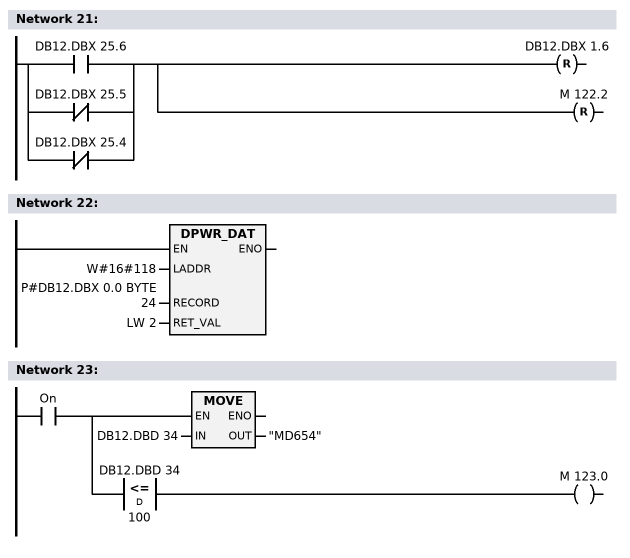
NETWORK
TITLE =
      O     DB12.DBX 25.6;
      ON    DB12.DBX 25.5;
      ON    DB12.DBX 25.4;
      R     DB12.DBX 1.6;
      R     M 122.2;
NETWORK
TITLE =
      CALL  "DPWR_DAT" (
           LADDR                    := W#16#118,
           RECORD                   := P#DB12.DBX 0.0 BYTE 24,
           RET_VAL                  := LW 2);
      NOP   0;
NETWORK
TITLE =
      A     "On";
      =     L 20.0;
      A     L 20.0;
      JNB   M019;
      L     DB12.DBD 34;
      T     "MD654";
M019: NOP   0;
      A     L 20.0;
      A(;
      L     DB12.DBD 34;
      L     100;
      <=D;
      );
      =     M 123.0;
END_FUNCTION

FUNCTION "FC50 - TEACH-IN" : VOID	// FC 50
VERSION : 0.1
BEGIN
// (block stored without names or comments; labels and parameter names are numbered)
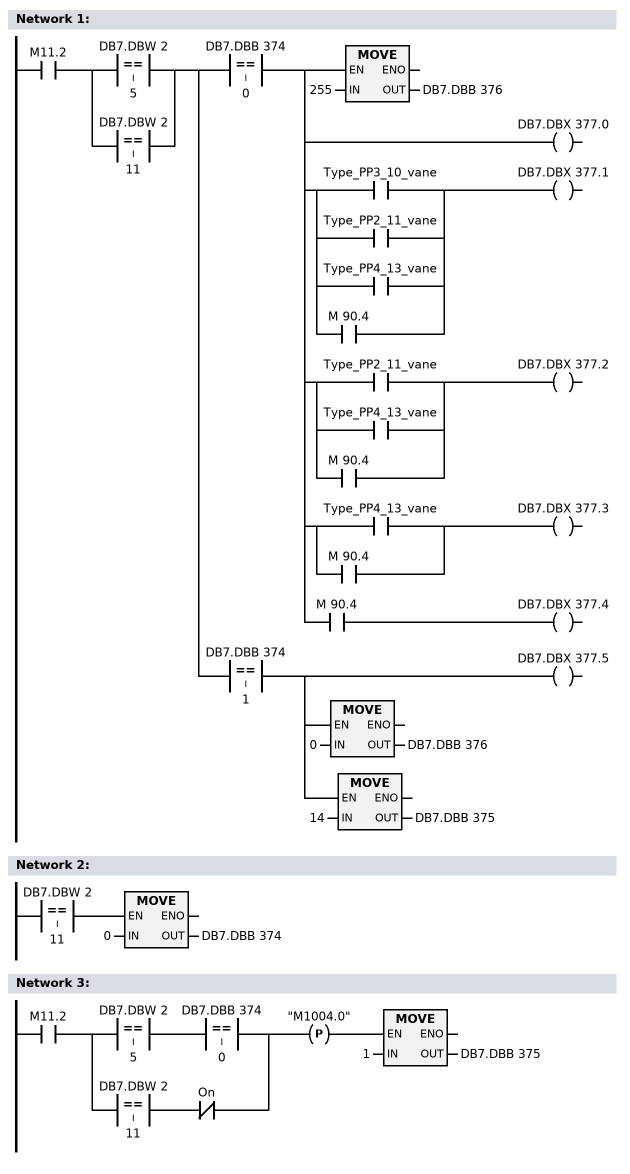
NETWORK
TITLE =
      A     "M11.2";
      A(;
      O(;
      L     DB7.DBW 2;
      L     5;
      ==I;
      );
      O(;
      L     DB7.DBW 2;
      L     11;
      ==I;
      );
      );
      =     L 8.0;
      A     L 8.0;
      A(;
      L     DB7.DBB 374;
      L     0;
      ==I;
      );
      =     L 8.1;
      A     L 8.1;
      JNB   M001;
      L     255;
      T     DB7.DBB 376;
M001: NOP   0;
      A     L 8.1;
      BLD   102;
      =     DB7.DBX 377.0;
      A     L 8.1;
      A(;
      O     "Type_PP3_10_vane";
      O     "Type_PP2_11_vane";
      O     "Type_PP4_13_vane";
      O     M 90.4;
      );
      =     DB7.DBX 377.1;
      A     L 8.1;
      A(;
      O     "Type_PP2_11_vane";
      O     "Type_PP4_13_vane";
      O     M 90.4;
      );
      =     DB7.DBX 377.2;
      A     L 8.1;
      A(;
      O     "Type_PP4_13_vane";
      O     M 90.4;
      );
      =     DB7.DBX 377.3;
      A     L 8.1;
      A     M 90.4;
      =     DB7.DBX 377.4;
      A     L 8.0;
      A(;
      L     DB7.DBB 374;
      L     1;
      ==I;
      );
      =     L 8.1;
      A     L 8.1;
      BLD   102;
      =     DB7.DBX 377.5;
      A     L 8.1;
      JNB   M002;
      L     0;
      T     DB7.DBB 376;
M002: NOP   0;
      A     L 8.1;
      JNB   M003;
      L     14;
      T     DB7.DBB 375;
M003: NOP   0;
NETWORK
TITLE =
      A(;
      L     DB7.DBW 2;
      L     11;
      ==I;
      );
      JNB   M004;
      L     0;
      T     DB7.DBB 374;
M004: NOP   0;
NETWORK
TITLE =
      A     "M11.2";
      A(;
      A(;
      L     DB7.DBW 2;
      L     5;
      ==I;
      );
      A(;
      L     DB7.DBB 374;
      L     0;
      ==I;
      );
      O;
      A(;
      L     DB7.DBW 2;
      L     11;
      ==I;
      );
      AN    "On";
      );
      FP    "M1004.0";
      JNB   M005;
      L     1;
      T     DB7.DBB 375;
M005: NOP   0;
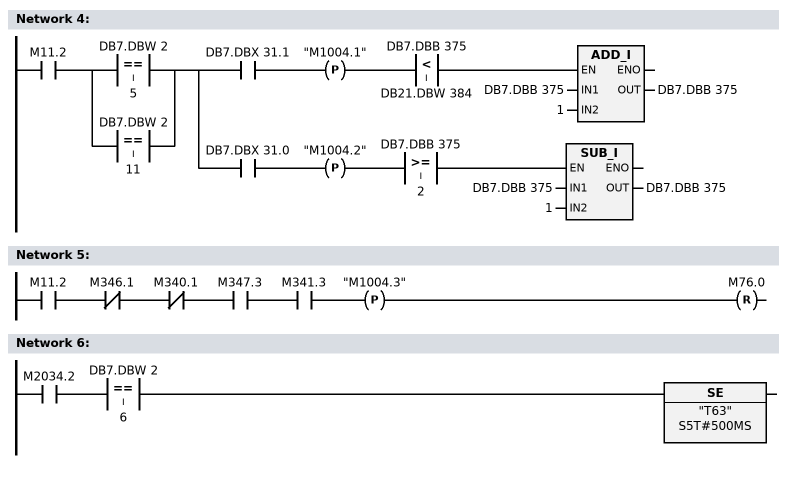
NETWORK
TITLE =
      A     "M11.2";
      A(;
      O(;
      L     DB7.DBW 2;
      L     5;
      ==I;
      );
      O(;
      L     DB7.DBW 2;
      L     11;
      ==I;
      );
      );
      =     L 8.0;
      A     L 8.0;
      A     DB7.DBX 31.1;
      FP    "M1004.1";
      A(;
      L     DB7.DBB 375;
      L     DB21.DBW 384;
      <I;
      );
      JNB   M006;
      L     DB7.DBB 375;
      L     1;
      +I;
      T     DB7.DBB 375;
M006: NOP   0;
      A     L 8.0;
      A     DB7.DBX 31.0;
      FP    "M1004.2";
      A(;
      L     DB7.DBB 375;
      L     2;
      >=I;
      );
      JNB   M007;
      L     DB7.DBB 375;
      L     1;
      -I;
      T     DB7.DBB 375;
M007: NOP   0;
NETWORK
TITLE =
      A     "M11.2";
      AN    "M346.1";
      AN    "M340.1";
      A     "M347.3";
      A     "M341.3";
      FP    "M1004.3";
      R     "M76.0";
NETWORK
TITLE =
      A     "M2034.2";
      A(;
      L     DB7.DBW 2;
      L     6;
      ==I;
      );
      L     S5T#500MS;
      SE    "T63";
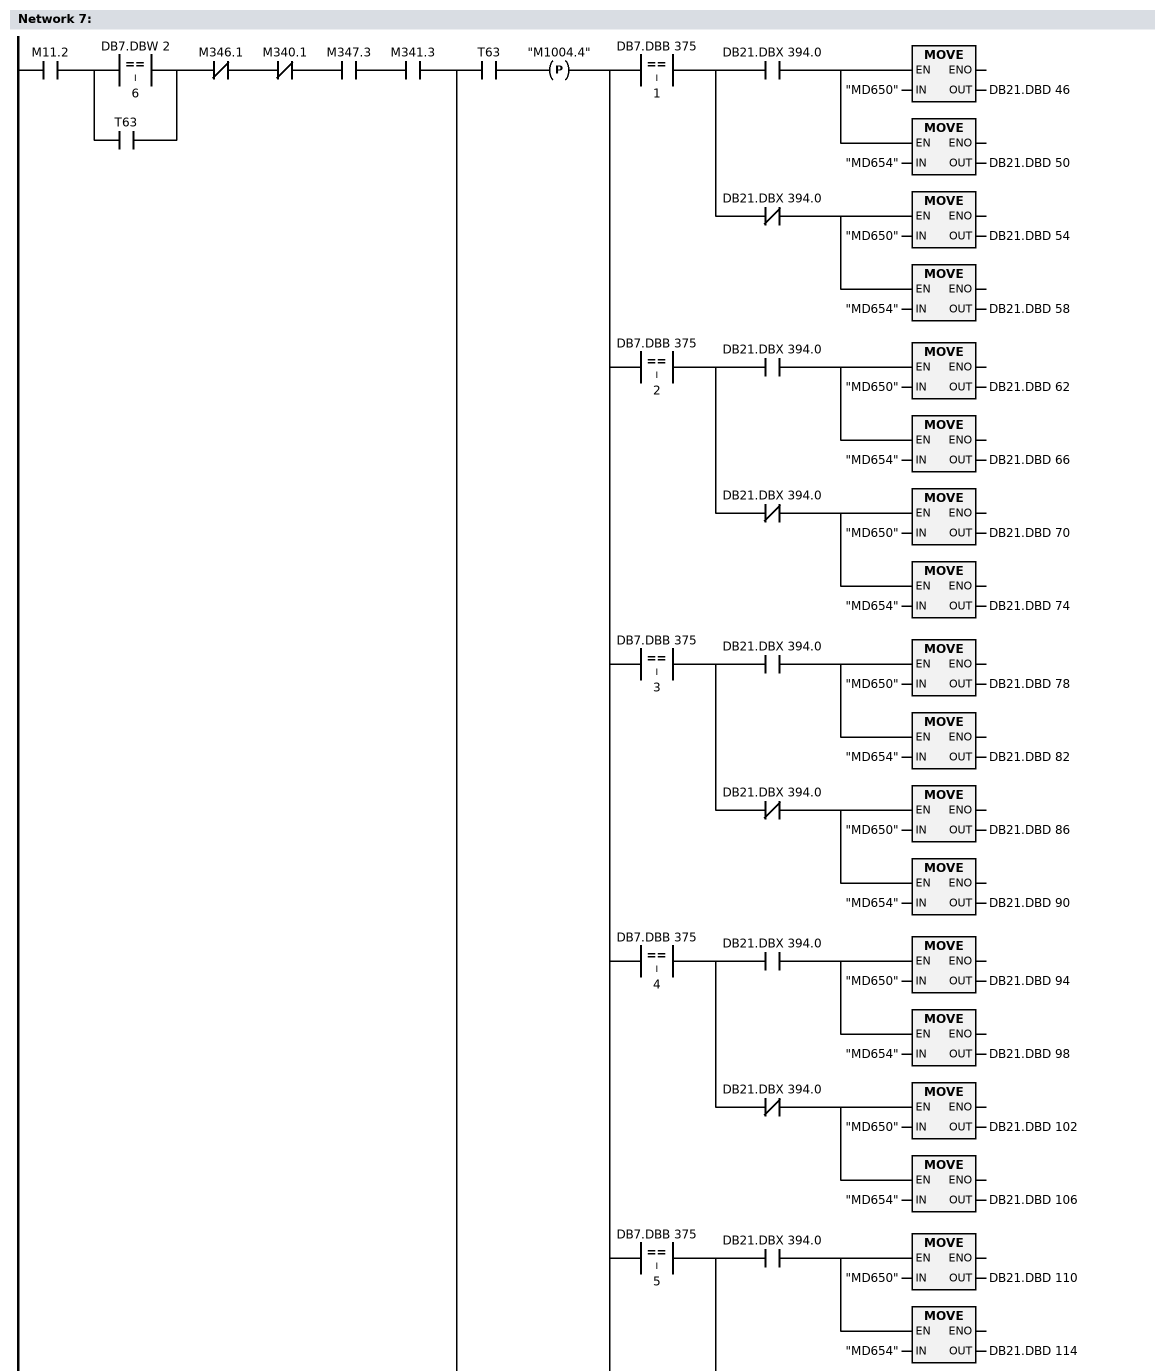
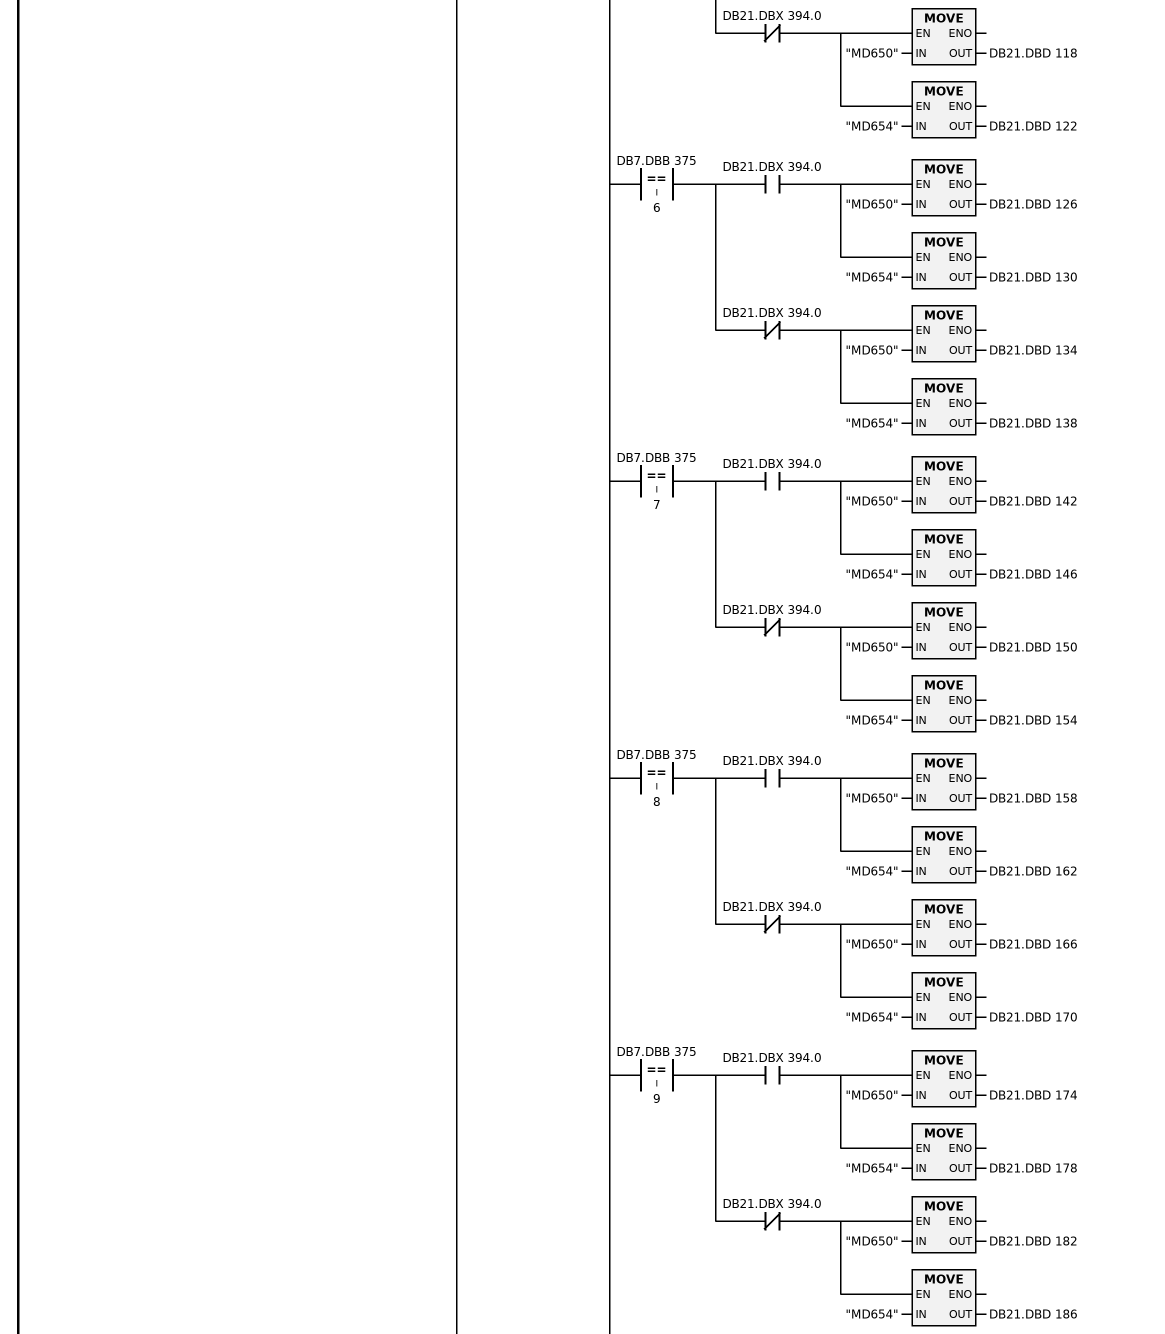
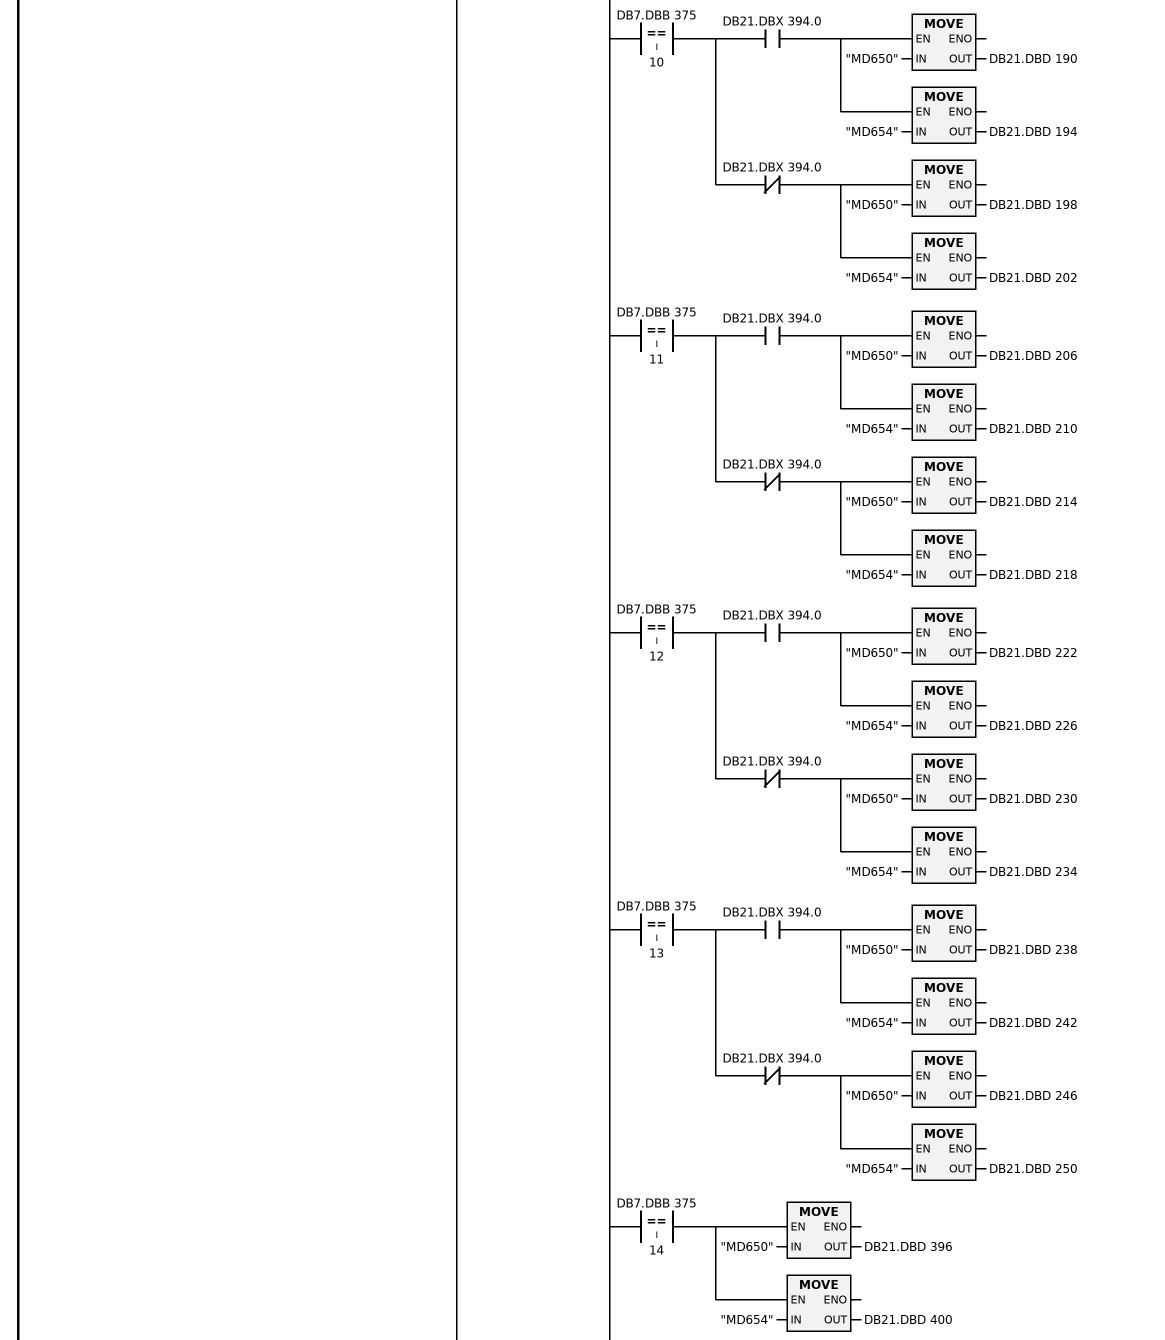
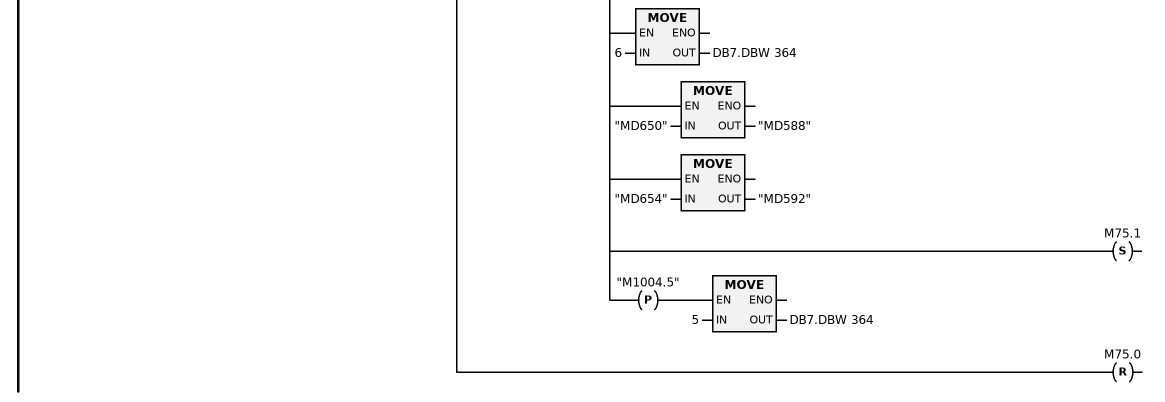
NETWORK
TITLE =
      A     "M11.2";
      A(;
      O(;
      L     DB7.DBW 2;
      L     6;
      ==I;
      );
      O     "T63";
      );
      AN    "M346.1";
      AN    "M340.1";
      A     "M347.3";
      A     "M341.3";
      =     L 8.0;
      A     L 8.0;
      A     "T63";
      FP    "M1004.4";
      =     L 8.1;
      A     L 8.1;
      A(;
      L     DB7.DBB 375;
      L     1;
      ==I;
      );
      =     L 8.2;
      A     L 8.2;
      A     DB21.DBX 394.0;
      =     L 8.3;
      A     L 8.3;
      JNB   M008;
      L     "MD650";
      T     DB21.DBD 46;
M008: NOP   0;
      A     L 8.3;
      JNB   M009;
      L     "MD654";
      T     DB21.DBD 50;
M009: NOP   0;
      A     L 8.2;
      AN    DB21.DBX 394.0;
      =     L 8.3;
      A     L 8.3;
      JNB   M010;
      L     "MD650";
      T     DB21.DBD 54;
M010: NOP   0;
      A     L 8.3;
      JNB   M011;
      L     "MD654";
      T     DB21.DBD 58;
M011: NOP   0;
      A     L 8.1;
      A(;
      L     DB7.DBB 375;
      L     2;
      ==I;
      );
      =     L 8.2;
      A     L 8.2;
      A     DB21.DBX 394.0;
      =     L 8.3;
      A     L 8.3;
      JNB   M012;
      L     "MD650";
      T     DB21.DBD 62;
M012: NOP   0;
      A     L 8.3;
      JNB   M013;
      L     "MD654";
      T     DB21.DBD 66;
M013: NOP   0;
      A     L 8.2;
      AN    DB21.DBX 394.0;
      =     L 8.3;
      A     L 8.3;
      JNB   M014;
      L     "MD650";
      T     DB21.DBD 70;
M014: NOP   0;
      A     L 8.3;
      JNB   M015;
      L     "MD654";
      T     DB21.DBD 74;
M015: NOP   0;
      A     L 8.1;
      A(;
      L     DB7.DBB 375;
      L     3;
      ==I;
      );
      =     L 8.2;
      A     L 8.2;
      A     DB21.DBX 394.0;
      =     L 8.3;
      A     L 8.3;
      JNB   M016;
      L     "MD650";
      T     DB21.DBD 78;
M016: NOP   0;
      A     L 8.3;
      JNB   M017;
      L     "MD654";
      T     DB21.DBD 82;
M017: NOP   0;
      A     L 8.2;
      AN    DB21.DBX 394.0;
      =     L 8.3;
      A     L 8.3;
      JNB   M018;
      L     "MD650";
      T     DB21.DBD 86;
M018: NOP   0;
      A     L 8.3;
      JNB   M019;
      L     "MD654";
      T     DB21.DBD 90;
M019: NOP   0;
      A     L 8.1;
      A(;
      L     DB7.DBB 375;
      L     4;
      ==I;
      );
      =     L 8.2;
      A     L 8.2;
      A     DB21.DBX 394.0;
      =     L 8.3;
      A     L 8.3;
      JNB   M020;
      L     "MD650";
      T     DB21.DBD 94;
M020: NOP   0;
      A     L 8.3;
      JNB   M021;
      L     "MD654";
      T     DB21.DBD 98;
M021: NOP   0;
      A     L 8.2;
      AN    DB21.DBX 394.0;
      =     L 8.3;
      A     L 8.3;
      JNB   M022;
      L     "MD650";
      T     DB21.DBD 102;
M022: NOP   0;
      A     L 8.3;
      JNB   M023;
      L     "MD654";
      T     DB21.DBD 106;
M023: NOP   0;
      A     L 8.1;
      A(;
      L     DB7.DBB 375;
      L     5;
      ==I;
      );
      =     L 8.2;
      A     L 8.2;
      A     DB21.DBX 394.0;
      =     L 8.3;
      A     L 8.3;
      JNB   M024;
      L     "MD650";
      T     DB21.DBD 110;
M024: NOP   0;
      A     L 8.3;
      JNB   M025;
      L     "MD654";
      T     DB21.DBD 114;
M025: NOP   0;
      A     L 8.2;
      AN    DB21.DBX 394.0;
      =     L 8.3;
      A     L 8.3;
      JNB   M026;
      L     "MD650";
      T     DB21.DBD 118;
M026: NOP   0;
      A     L 8.3;
      JNB   M027;
      L     "MD654";
      T     DB21.DBD 122;
M027: NOP   0;
      A     L 8.1;
      A(;
      L     DB7.DBB 375;
      L     6;
      ==I;
      );
      =     L 8.2;
      A     L 8.2;
      A     DB21.DBX 394.0;
      =     L 8.3;
      A     L 8.3;
      JNB   M028;
      L     "MD650";
      T     DB21.DBD 126;
M028: NOP   0;
      A     L 8.3;
      JNB   M029;
      L     "MD654";
      T     DB21.DBD 130;
M029: NOP   0;
      A     L 8.2;
      AN    DB21.DBX 394.0;
      =     L 8.3;
      A     L 8.3;
      JNB   M030;
      L     "MD650";
      T     DB21.DBD 134;
M030: NOP   0;
      A     L 8.3;
      JNB   M031;
      L     "MD654";
      T     DB21.DBD 138;
M031: NOP   0;
      A     L 8.1;
      A(;
      L     DB7.DBB 375;
      L     7;
      ==I;
      );
      =     L 8.2;
      A     L 8.2;
      A     DB21.DBX 394.0;
      =     L 8.3;
      A     L 8.3;
      JNB   M032;
      L     "MD650";
      T     DB21.DBD 142;
M032: NOP   0;
      A     L 8.3;
      JNB   M033;
      L     "MD654";
      T     DB21.DBD 146;
M033: NOP   0;
      A     L 8.2;
      AN    DB21.DBX 394.0;
      =     L 8.3;
      A     L 8.3;
      JNB   M034;
      L     "MD650";
      T     DB21.DBD 150;
M034: NOP   0;
      A     L 8.3;
      JNB   M035;
      L     "MD654";
      T     DB21.DBD 154;
M035: NOP   0;
      A     L 8.1;
      A(;
      L     DB7.DBB 375;
      L     8;
      ==I;
      );
      =     L 8.2;
      A     L 8.2;
      A     DB21.DBX 394.0;
      =     L 8.3;
      A     L 8.3;
      JNB   M036;
      L     "MD650";
      T     DB21.DBD 158;
M036: NOP   0;
      A     L 8.3;
      JNB   M037;
      L     "MD654";
      T     DB21.DBD 162;
M037: NOP   0;
      A     L 8.2;
      AN    DB21.DBX 394.0;
      =     L 8.3;
      A     L 8.3;
      JNB   M038;
      L     "MD650";
      T     DB21.DBD 166;
M038: NOP   0;
      A     L 8.3;
      JNB   M039;
      L     "MD654";
      T     DB21.DBD 170;
M039: NOP   0;
      A     L 8.1;
      A(;
      L     DB7.DBB 375;
      L     9;
      ==I;
      );
      =     L 8.2;
      A     L 8.2;
      A     DB21.DBX 394.0;
      =     L 8.3;
      A     L 8.3;
      JNB   M040;
      L     "MD650";
      T     DB21.DBD 174;
M040: NOP   0;
      A     L 8.3;
      JNB   M041;
      L     "MD654";
      T     DB21.DBD 178;
M041: NOP   0;
      A     L 8.2;
      AN    DB21.DBX 394.0;
      =     L 8.3;
      A     L 8.3;
      JNB   M042;
      L     "MD650";
      T     DB21.DBD 182;
M042: NOP   0;
      A     L 8.3;
      JNB   M043;
      L     "MD654";
      T     DB21.DBD 186;
M043: NOP   0;
      A     L 8.1;
      A(;
      L     DB7.DBB 375;
      L     10;
      ==I;
      );
      =     L 8.2;
      A     L 8.2;
      A     DB21.DBX 394.0;
      =     L 8.3;
      A     L 8.3;
      JNB   M044;
      L     "MD650";
      T     DB21.DBD 190;
M044: NOP   0;
      A     L 8.3;
      JNB   M045;
      L     "MD654";
      T     DB21.DBD 194;
M045: NOP   0;
      A     L 8.2;
      AN    DB21.DBX 394.0;
      =     L 8.3;
      A     L 8.3;
      JNB   M046;
      L     "MD650";
      T     DB21.DBD 198;
M046: NOP   0;
      A     L 8.3;
      JNB   M047;
      L     "MD654";
      T     DB21.DBD 202;
M047: NOP   0;
      A     L 8.1;
      A(;
      L     DB7.DBB 375;
      L     11;
      ==I;
      );
      =     L 8.2;
      A     L 8.2;
      A     DB21.DBX 394.0;
      =     L 8.3;
      A     L 8.3;
      JNB   M048;
      L     "MD650";
      T     DB21.DBD 206;
M048: NOP   0;
      A     L 8.3;
      JNB   M049;
      L     "MD654";
      T     DB21.DBD 210;
M049: NOP   0;
      A     L 8.2;
      AN    DB21.DBX 394.0;
      =     L 8.3;
      A     L 8.3;
      JNB   M050;
      L     "MD650";
      T     DB21.DBD 214;
M050: NOP   0;
      A     L 8.3;
      JNB   M051;
      L     "MD654";
      T     DB21.DBD 218;
M051: NOP   0;
      A     L 8.1;
      A(;
      L     DB7.DBB 375;
      L     12;
      ==I;
      );
      =     L 8.2;
      A     L 8.2;
      A     DB21.DBX 394.0;
      =     L 8.3;
      A     L 8.3;
      JNB   M052;
      L     "MD650";
      T     DB21.DBD 222;
M052: NOP   0;
      A     L 8.3;
      JNB   M053;
      L     "MD654";
      T     DB21.DBD 226;
M053: NOP   0;
      A     L 8.2;
      AN    DB21.DBX 394.0;
      =     L 8.3;
      A     L 8.3;
      JNB   M054;
      L     "MD650";
      T     DB21.DBD 230;
M054: NOP   0;
      A     L 8.3;
      JNB   M055;
      L     "MD654";
      T     DB21.DBD 234;
M055: NOP   0;
      A     L 8.1;
      A(;
      L     DB7.DBB 375;
      L     13;
      ==I;
      );
      =     L 8.2;
      A     L 8.2;
      A     DB21.DBX 394.0;
      =     L 8.3;
      A     L 8.3;
      JNB   M056;
      L     "MD650";
      T     DB21.DBD 238;
M056: NOP   0;
      A     L 8.3;
      JNB   M057;
      L     "MD654";
      T     DB21.DBD 242;
M057: NOP   0;
      A     L 8.2;
      AN    DB21.DBX 394.0;
      =     L 8.3;
      A     L 8.3;
      JNB   M058;
      L     "MD650";
      T     DB21.DBD 246;
M058: NOP   0;
      A     L 8.3;
      JNB   M059;
      L     "MD654";
      T     DB21.DBD 250;
M059: NOP   0;
      A     L 8.1;
      A(;
      L     DB7.DBB 375;
      L     14;
      ==I;
      );
      =     L 8.2;
      A     L 8.2;
      JNB   M060;
      L     "MD650";
      T     DB21.DBD 396;
M060: NOP   0;
      A     L 8.2;
      JNB   M061;
      L     "MD654";
      T     DB21.DBD 400;
M061: NOP   0;
      A     L 8.1;
      JNB   M062;
      L     6;
      T     DB7.DBW 364;
M062: NOP   0;
      A     L 8.1;
      JNB   M063;
      L     "MD650";
      T     "MD588";
M063: NOP   0;
      A     L 8.1;
      JNB   M064;
      L     "MD654";
      T     "MD592";
M064: NOP   0;
      A     L 8.1;
      BLD   102;
      S     "M75.1";
      A     L 8.1;
      FP    "M1004.5";
      JNB   M065;
      L     5;
      T     DB7.DBW 364;
M065: NOP   0;
      A     L 8.0;
      BLD   102;
      R     "M75.0";
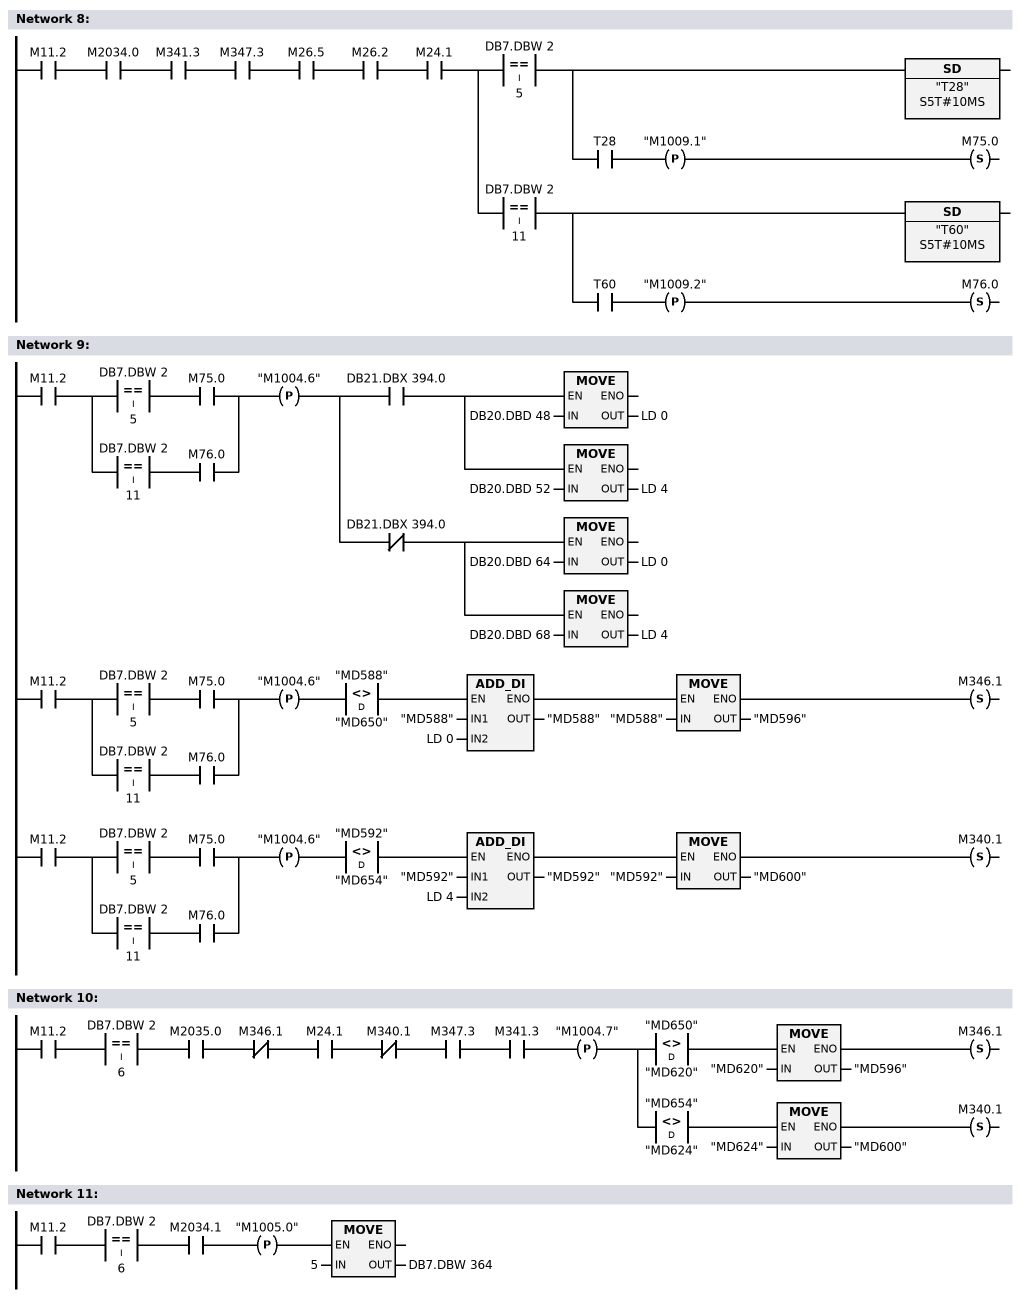
NETWORK
TITLE =
      A     "M11.2";
      A     "M2034.0";
      A     "M341.3";
      A     "M347.3";
      A     "M26.5";
      A     "M26.2";
      A     "M24.1";
      =     L 8.0;
      A     L 8.0;
      A(;
      L     DB7.DBW 2;
      L     5;
      ==I;
      );
      =     L 8.1;
      A     L 8.1;
      BLD   102;
      L     S5T#10MS;
      SD    "T28";
      A     L 8.1;
      A     "T28";
      FP    "M1009.1";
      S     "M75.0";
      A     L 8.0;
      A(;
      L     DB7.DBW 2;
      L     11;
      ==I;
      );
      =     L 8.1;
      A     L 8.1;
      BLD   102;
      L     S5T#10MS;
      SD    "T60";
      A     L 8.1;
      A     "T60";
      FP    "M1009.2";
      S     "M76.0";
NETWORK
TITLE =
      A     "M11.2";
      A(;
      A(;
      L     DB7.DBW 2;
      L     5;
      ==I;
      );
      A     "M75.0";
      O;
      A(;
      L     DB7.DBW 2;
      L     11;
      ==I;
      );
      A     "M76.0";
      );
      FP    "M1004.6";
      =     L 8.0;
      A     L 8.0;
      A     DB21.DBX 394.0;
      =     L 8.1;
      A     L 8.1;
      JNB   M066;
      L     DB20.DBD 48;
      T     LD 0;
M066: NOP   0;
      A     L 8.1;
      JNB   M067;
      L     DB20.DBD 52;
      T     LD 4;
M067: NOP   0;
      A     L 8.0;
      AN    DB21.DBX 394.0;
      =     L 8.1;
      A     L 8.1;
      JNB   M068;
      L     DB20.DBD 64;
      T     LD 0;
M068: NOP   0;
      A     L 8.1;
      JNB   M069;
      L     DB20.DBD 68;
      T     LD 4;
M069: NOP   0;
      A(;
      A     L 8.0;
      A(;
      L     "MD588";
      L     "MD650";
      <>D;
      );
      JNB   M070;
      L     "MD588";
      L     LD 0;
      +D;
      T     "MD588";
      AN    OV;
      SAVE;
      CLR;
M070: A     BR;
      );
      JNB   M071;
      L     "MD588";
      T     "MD596";
      SET;
      SAVE;
      CLR;
M071: A     BR;
      S     "M346.1";
      A(;
      A     L 8.0;
      A(;
      L     "MD592";
      L     "MD654";
      <>D;
      );
      JNB   M072;
      L     "MD592";
      L     LD 4;
      +D;
      T     "MD592";
      AN    OV;
      SAVE;
      CLR;
M072: A     BR;
      );
      JNB   M073;
      L     "MD592";
      T     "MD600";
      SET;
      SAVE;
      CLR;
M073: A     BR;
      S     "M340.1";
NETWORK
TITLE =
      A     "M11.2";
      A(;
      L     DB7.DBW 2;
      L     6;
      ==I;
      );
      A     "M2035.0";
      AN    "M346.1";
      A     "M24.1";
      AN    "M340.1";
      A     "M347.3";
      A     "M341.3";
      FP    "M1004.7";
      =     L 8.0;
      A     L 8.0;
      A(;
      L     "MD650";
      L     "MD620";
      <>D;
      );
      JNB   M074;
      L     "MD620";
      T     "MD596";
      SET;
      SAVE;
      CLR;
M074: A     BR;
      S     "M346.1";
      A     L 8.0;
      A(;
      L     "MD654";
      L     "MD624";
      <>D;
      );
      JNB   M075;
      L     "MD624";
      T     "MD600";
      SET;
      SAVE;
      CLR;
M075: A     BR;
      S     "M340.1";
NETWORK
TITLE =
      A     "M11.2";
      A(;
      L     DB7.DBW 2;
      L     6;
      ==I;
      );
      A     "M2034.1";
      FP    "M1005.0";
      JNB   M076;
      L     5;
      T     DB7.DBW 364;
M076: NOP   0;
END_FUNCTION

FUNCTION "FC51 - TYPE TOOL" : VOID	// FC 51
VERSION : 0.1
BEGIN
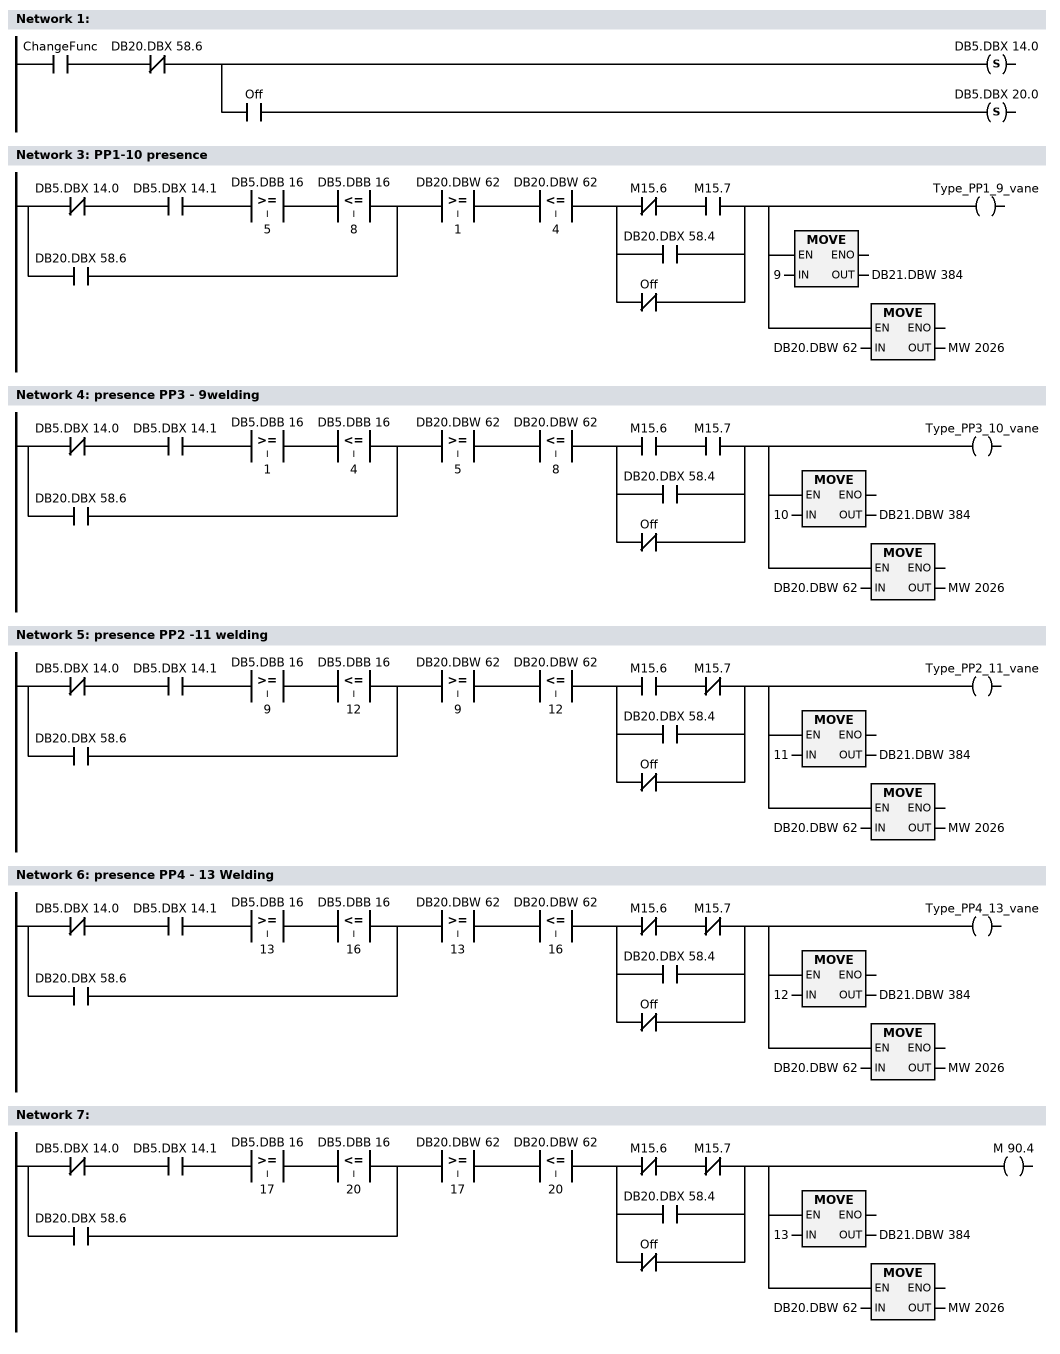
NETWORK
TITLE =
      A     "ChangeFunc";
      AN    DB20.DBX 58.6;
      =     L 0.0;
      A     L 0.0;
      BLD   102;
      S     DB5.DBX 14.0;
      A     L 0.0;
      A     "Off";
      S     DB5.DBX 20.0;
NETWORK
TITLE =
NETWORK
TITLE = PP1-10 presence
      A(;
      AN    DB5.DBX 14.0;
      A     DB5.DBX 14.1;
      A(;
      L     DB5.DBB 16;
      L     5;
      >=I;
      );
      A(;
      L     DB5.DBB 16;
      L     8;
      <=I;
      );
      O     DB20.DBX 58.6;
      );
      A(;
      L     DB20.DBW 62;
      L     1;
      >=I;
      );
      A(;
      L     DB20.DBW 62;
      L     4;
      <=I;
      );
      A(;
      AN    "M15.6";
      A     "M15.7";
      O     DB20.DBX 58.4;
      ON    "Off";
      );
      =     L 0.0;
      A     L 0.0;
      BLD   102;
      =     "Type_PP1_9_vane";
      A     L 0.0;
      JNB   _001;
      L     9;
      T     DB21.DBW 384;
_001: NOP   0;
      A     L 0.0;
      JNB   _002;
      L     DB20.DBW 62;
      T     MW 2026;
_002: NOP   0;
NETWORK
TITLE = presence PP3 - 9welding
      A(;
      AN    DB5.DBX 14.0;
      A     DB5.DBX 14.1;
      A(;
      L     DB5.DBB 16;
      L     1;
      >=I;
      );
      A(;
      L     DB5.DBB 16;
      L     4;
      <=I;
      );
      O     DB20.DBX 58.6;
      );
      A(;
      L     DB20.DBW 62;
      L     5;
      >=I;
      );
      A(;
      L     DB20.DBW 62;
      L     8;
      <=I;
      );
      A(;
      A     "M15.6";
      A     "M15.7";
      O     DB20.DBX 58.4;
      ON    "Off";
      );
      =     L 0.0;
      A     L 0.0;
      BLD   102;
      =     "Type_PP3_10_vane";
      A     L 0.0;
      JNB   _003;
      L     10;
      T     DB21.DBW 384;
_003: NOP   0;
      A     L 0.0;
      JNB   _004;
      L     DB20.DBW 62;
      T     MW 2026;
_004: NOP   0;
NETWORK
TITLE = presence PP2 -11 welding
      A(;
      AN    DB5.DBX 14.0;
      A     DB5.DBX 14.1;
      A(;
      L     DB5.DBB 16;
      L     9;
      >=I;
      );
      A(;
      L     DB5.DBB 16;
      L     12;
      <=I;
      );
      O     DB20.DBX 58.6;
      );
      A(;
      L     DB20.DBW 62;
      L     9;
      >=I;
      );
      A(;
      L     DB20.DBW 62;
      L     12;
      <=I;
      );
      A(;
      A     "M15.6";
      AN    "M15.7";
      O     DB20.DBX 58.4;
      ON    "Off";
      );
      =     L 0.0;
      A     L 0.0;
      BLD   102;
      =     "Type_PP2_11_vane";
      A     L 0.0;
      JNB   _005;
      L     11;
      T     DB21.DBW 384;
_005: NOP   0;
      A     L 0.0;
      JNB   _006;
      L     DB20.DBW 62;
      T     MW 2026;
_006: NOP   0;
NETWORK
TITLE = presence PP4 - 13 Welding
      A(;
      AN    DB5.DBX 14.0;
      A     DB5.DBX 14.1;
      A(;
      L     DB5.DBB 16;
      L     13;
      >=I;
      );
      A(;
      L     DB5.DBB 16;
      L     16;
      <=I;
      );
      O     DB20.DBX 58.6;
      );
      A(;
      L     DB20.DBW 62;
      L     13;
      >=I;
      );
      A(;
      L     DB20.DBW 62;
      L     16;
      <=I;
      );
      A(;
      AN    "M15.6";
      AN    "M15.7";
      O     DB20.DBX 58.4;
      ON    "Off";
      );
      =     L 0.0;
      A     L 0.0;
      BLD   102;
      =     "Type_PP4_13_vane";
      A     L 0.0;
      JNB   _007;
      L     12;
      T     DB21.DBW 384;
_007: NOP   0;
      A     L 0.0;
      JNB   _008;
      L     DB20.DBW 62;
      T     MW 2026;
_008: NOP   0;
NETWORK
TITLE =
      A(;
      AN    DB5.DBX 14.0;
      A     DB5.DBX 14.1;
      A(;
      L     DB5.DBB 16;
      L     17;
      >=I;
      );
      A(;
      L     DB5.DBB 16;
      L     20;
      <=I;
      );
      O     DB20.DBX 58.6;
      );
      A(;
      L     DB20.DBW 62;
      L     17;
      >=I;
      );
      A(;
      L     DB20.DBW 62;
      L     20;
      <=I;
      );
      A(;
      AN    "M15.6";
      AN    "M15.7";
      O     DB20.DBX 58.4;
      ON    "Off";
      );
      =     L 0.0;
      A     L 0.0;
      BLD   102;
      =     M 90.4;
      A     L 0.0;
      JNB   _009;
      L     13;
      T     DB21.DBW 384;
_009: NOP   0;
      A     L 0.0;
      JNB   _00a;
      L     DB20.DBW 62;
      T     MW 2026;
_00a: NOP   0;
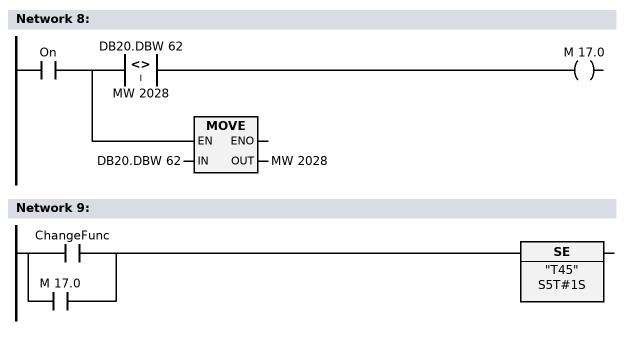
NETWORK
TITLE =
      A     "On";
      =     L 0.0;
      A     L 0.0;
      A(;
      L     DB20.DBW 62;
      L     MW 2028;
      <>I;
      );
      =     M 17.0;
      A     L 0.0;
      JNB   _00b;
      L     DB20.DBW 62;
      T     MW 2028;
_00b: NOP   0;
NETWORK
TITLE =
      O     "ChangeFunc";
      O     M 17.0;
      L     S5T#1S;
      SE    "T45";
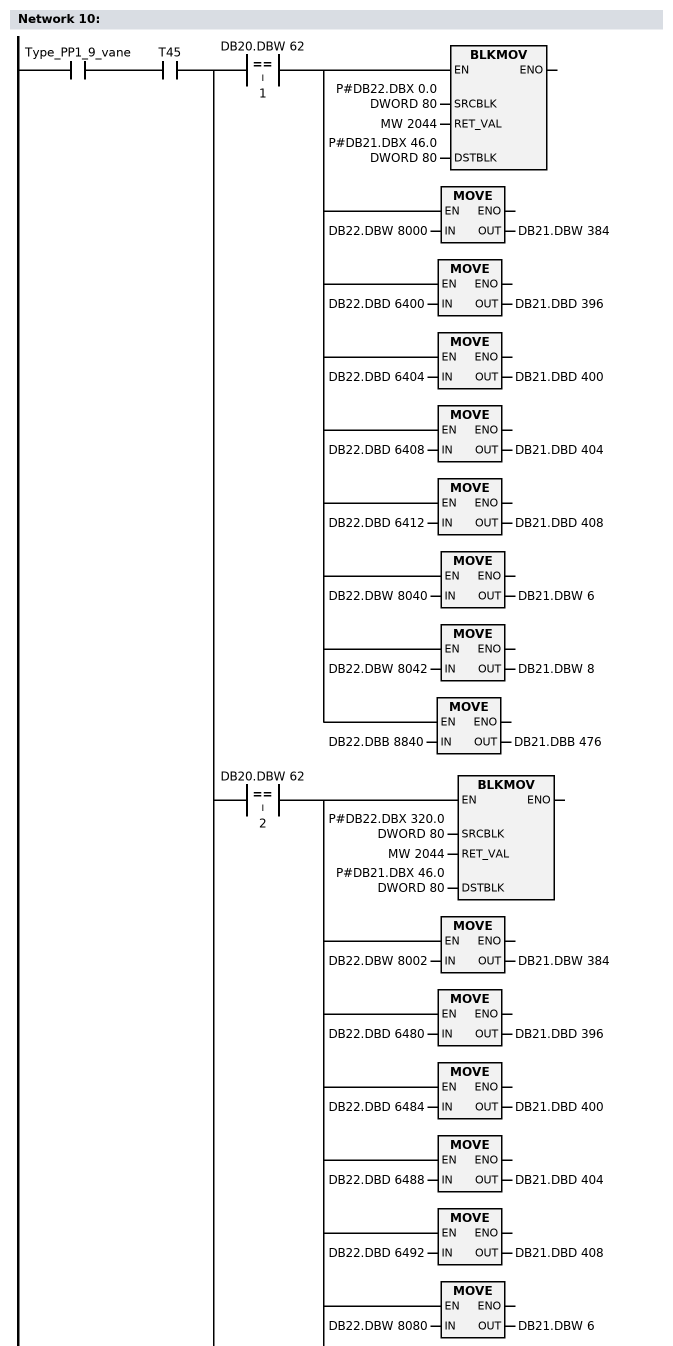
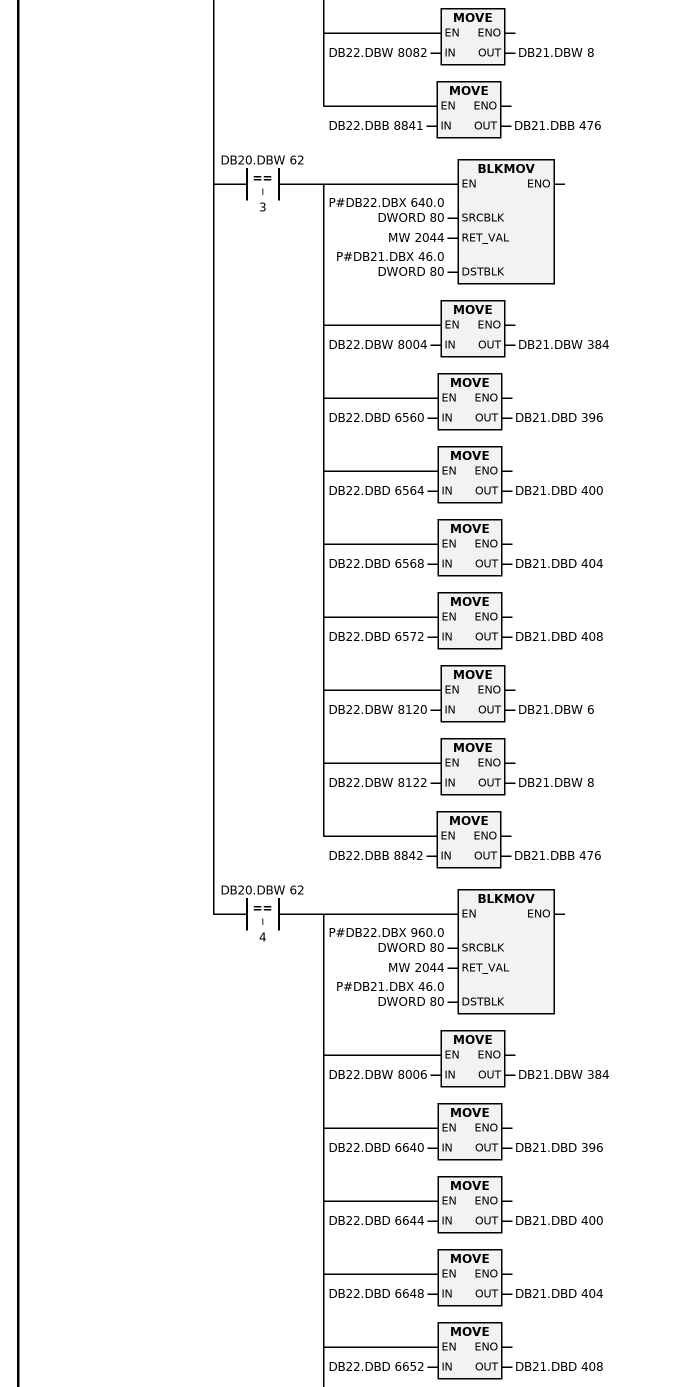
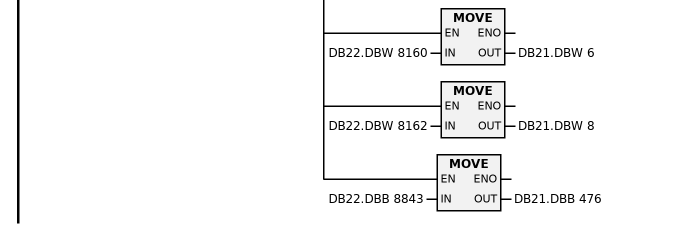
NETWORK
TITLE =
      A     "Type_PP1_9_vane";
      A     "T45";
      =     L 0.0;
      A     L 0.0;
      A(;
      L     DB20.DBW 62;
      L     1;
      ==I;
      );
      =     L 0.1;
      A     L 0.1;
      JNB   _00c;
      CALL  "BLKMOV" (
           SRCBLK                   := P#DB22.DBX 0.0 DWORD 80,
           RET_VAL                  := MW 2044,
           DSTBLK                   := P#DB21.DBX 46.0 DWORD 80);
_00c: NOP   0;
      A     L 0.1;
      JNB   _00d;
      L     DB22.DBW 8000;
      T     DB21.DBW 384;
_00d: NOP   0;
      A     L 0.1;
      JNB   _00e;
      L     DB22.DBD 6400;
      T     DB21.DBD 396;
_00e: NOP   0;
      A     L 0.1;
      JNB   _00f;
      L     DB22.DBD 6404;
      T     DB21.DBD 400;
_00f: NOP   0;
      A     L 0.1;
      JNB   _010;
      L     DB22.DBD 6408;
      T     DB21.DBD 404;
_010: NOP   0;
      A     L 0.1;
      JNB   _011;
      L     DB22.DBD 6412;
      T     DB21.DBD 408;
_011: NOP   0;
      A     L 0.1;
      JNB   _012;
      L     DB22.DBW 8040;
      T     DB21.DBW 6;
_012: NOP   0;
      A     L 0.1;
      JNB   _013;
      L     DB22.DBW 8042;
      T     DB21.DBW 8;
_013: NOP   0;
      A     L 0.1;
      JNB   _014;
      L     DB22.DBB 8840;
      T     DB21.DBB 476;
_014: NOP   0;
      A     L 0.0;
      A(;
      L     DB20.DBW 62;
      L     2;
      ==I;
      );
      =     L 0.1;
      A     L 0.1;
      JNB   _015;
      CALL  "BLKMOV" (
           SRCBLK                   := P#DB22.DBX 320.0 DWORD 80,
           RET_VAL                  := MW 2044,
           DSTBLK                   := P#DB21.DBX 46.0 DWORD 80);
_015: NOP   0;
      A     L 0.1;
      JNB   _016;
      L     DB22.DBW 8002;
      T     DB21.DBW 384;
_016: NOP   0;
      A     L 0.1;
      JNB   _017;
      L     DB22.DBD 6480;
      T     DB21.DBD 396;
_017: NOP   0;
      A     L 0.1;
      JNB   _018;
      L     DB22.DBD 6484;
      T     DB21.DBD 400;
_018: NOP   0;
      A     L 0.1;
      JNB   _019;
      L     DB22.DBD 6488;
      T     DB21.DBD 404;
_019: NOP   0;
      A     L 0.1;
      JNB   _01a;
      L     DB22.DBD 6492;
      T     DB21.DBD 408;
_01a: NOP   0;
      A     L 0.1;
      JNB   _01b;
      L     DB22.DBW 8080;
      T     DB21.DBW 6;
_01b: NOP   0;
      A     L 0.1;
      JNB   _01c;
      L     DB22.DBW 8082;
      T     DB21.DBW 8;
_01c: NOP   0;
      A     L 0.1;
      JNB   _01d;
      L     DB22.DBB 8841;
      T     DB21.DBB 476;
_01d: NOP   0;
      A     L 0.0;
      A(;
      L     DB20.DBW 62;
      L     3;
      ==I;
      );
      =     L 0.1;
      A     L 0.1;
      JNB   _01e;
      CALL  "BLKMOV" (
           SRCBLK                   := P#DB22.DBX 640.0 DWORD 80,
           RET_VAL                  := MW 2044,
           DSTBLK                   := P#DB21.DBX 46.0 DWORD 80);
_01e: NOP   0;
      A     L 0.1;
      JNB   _01f;
      L     DB22.DBW 8004;
      T     DB21.DBW 384;
_01f: NOP   0;
      A     L 0.1;
      JNB   _020;
      L     DB22.DBD 6560;
      T     DB21.DBD 396;
_020: NOP   0;
      A     L 0.1;
      JNB   _021;
      L     DB22.DBD 6564;
      T     DB21.DBD 400;
_021: NOP   0;
      A     L 0.1;
      JNB   _022;
      L     DB22.DBD 6568;
      T     DB21.DBD 404;
_022: NOP   0;
      A     L 0.1;
      JNB   _023;
      L     DB22.DBD 6572;
      T     DB21.DBD 408;
_023: NOP   0;
      A     L 0.1;
      JNB   _024;
      L     DB22.DBW 8120;
      T     DB21.DBW 6;
_024: NOP   0;
      A     L 0.1;
      JNB   _025;
      L     DB22.DBW 8122;
      T     DB21.DBW 8;
_025: NOP   0;
      A     L 0.1;
      JNB   _026;
      L     DB22.DBB 8842;
      T     DB21.DBB 476;
_026: NOP   0;
      A     L 0.0;
      A(;
      L     DB20.DBW 62;
      L     4;
      ==I;
      );
      =     L 0.1;
      A     L 0.1;
      JNB   _027;
      CALL  "BLKMOV" (
           SRCBLK                   := P#DB22.DBX 960.0 DWORD 80,
           RET_VAL                  := MW 2044,
           DSTBLK                   := P#DB21.DBX 46.0 DWORD 80);
_027: NOP   0;
      A     L 0.1;
      JNB   _028;
      L     DB22.DBW 8006;
      T     DB21.DBW 384;
_028: NOP   0;
      A     L 0.1;
      JNB   _029;
      L     DB22.DBD 6640;
      T     DB21.DBD 396;
_029: NOP   0;
      A     L 0.1;
      JNB   _02a;
      L     DB22.DBD 6644;
      T     DB21.DBD 400;
_02a: NOP   0;
      A     L 0.1;
      JNB   _02b;
      L     DB22.DBD 6648;
      T     DB21.DBD 404;
_02b: NOP   0;
      A     L 0.1;
      JNB   _02c;
      L     DB22.DBD 6652;
      T     DB21.DBD 408;
_02c: NOP   0;
      A     L 0.1;
      JNB   _02d;
      L     DB22.DBW 8160;
      T     DB21.DBW 6;
_02d: NOP   0;
      A     L 0.1;
      JNB   _02e;
      L     DB22.DBW 8162;
      T     DB21.DBW 8;
_02e: NOP   0;
      A     L 0.1;
      JNB   _02f;
      L     DB22.DBB 8843;
      T     DB21.DBB 476;
_02f: NOP   0;
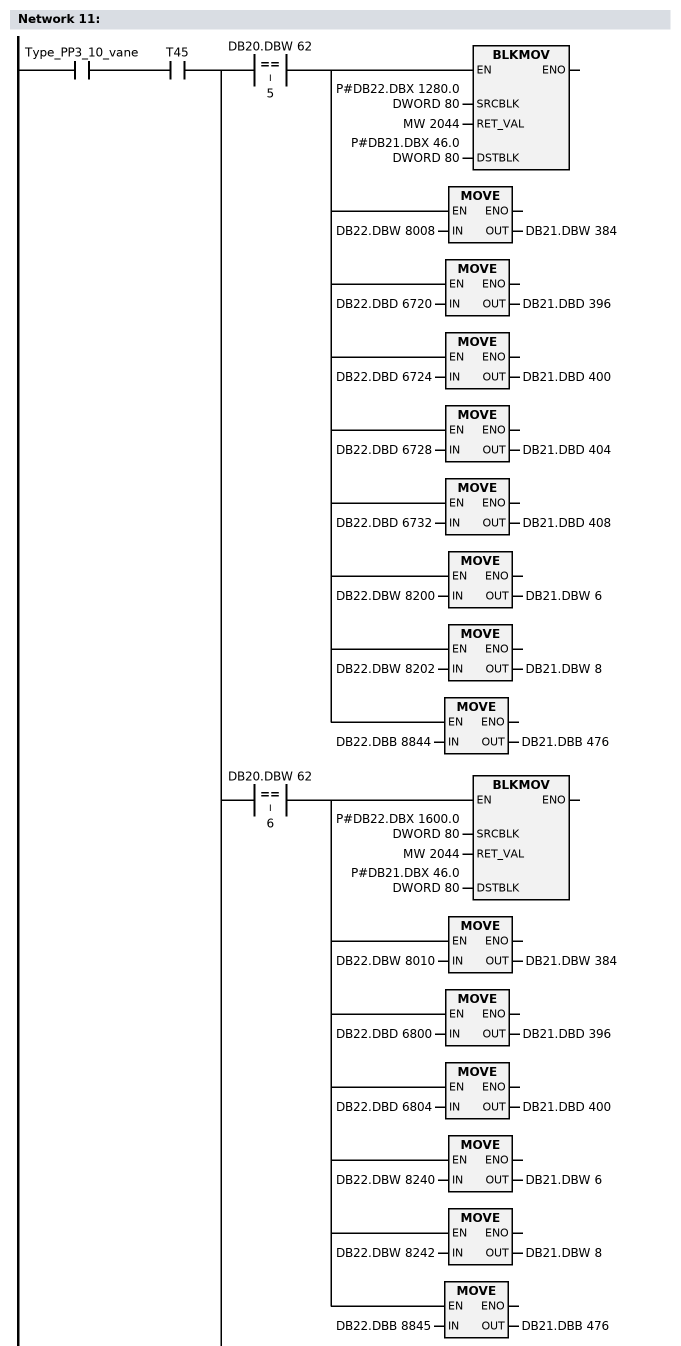
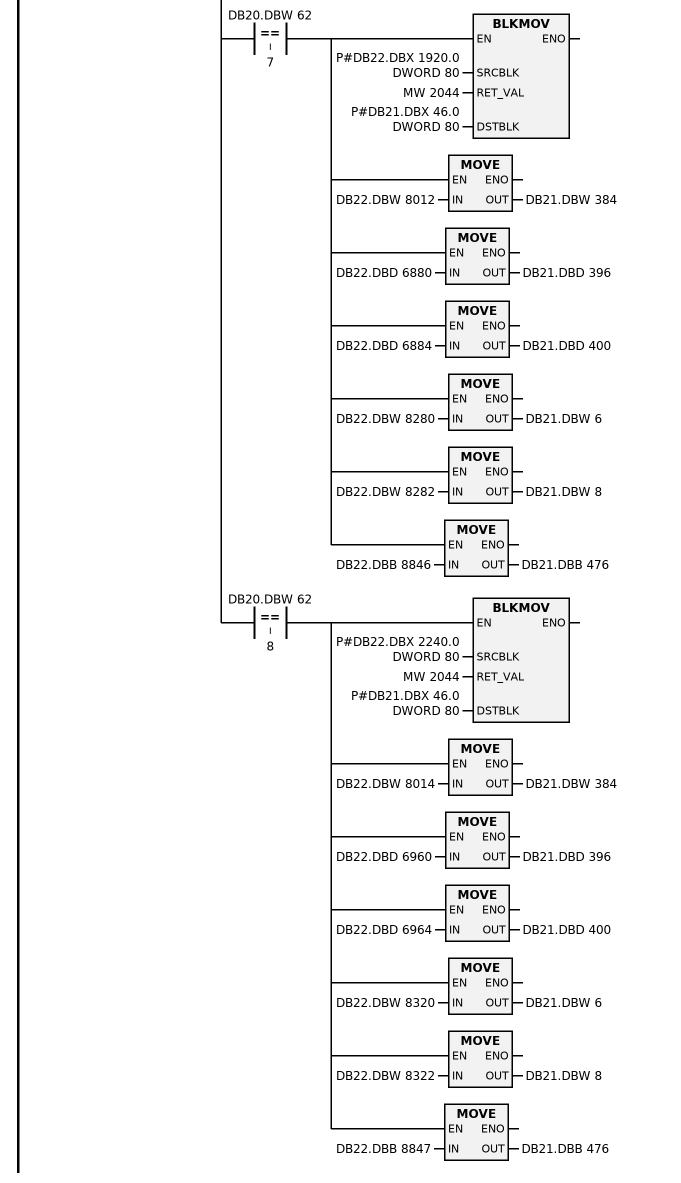
NETWORK
TITLE =
      A     "Type_PP3_10_vane";
      A     "T45";
      =     L 0.0;
      A     L 0.0;
      A(;
      L     DB20.DBW 62;
      L     5;
      ==I;
      );
      =     L 0.1;
      A     L 0.1;
      JNB   _030;
      CALL  "BLKMOV" (
           SRCBLK                   := P#DB22.DBX 1280.0 DWORD 80,
           RET_VAL                  := MW 2044,
           DSTBLK                   := P#DB21.DBX 46.0 DWORD 80);
_030: NOP   0;
      A     L 0.1;
      JNB   _031;
      L     DB22.DBW 8008;
      T     DB21.DBW 384;
_031: NOP   0;
      A     L 0.1;
      JNB   _032;
      L     DB22.DBD 6720;
      T     DB21.DBD 396;
_032: NOP   0;
      A     L 0.1;
      JNB   _033;
      L     DB22.DBD 6724;
      T     DB21.DBD 400;
_033: NOP   0;
      A     L 0.1;
      JNB   _034;
      L     DB22.DBD 6728;
      T     DB21.DBD 404;
_034: NOP   0;
      A     L 0.1;
      JNB   _035;
      L     DB22.DBD 6732;
      T     DB21.DBD 408;
_035: NOP   0;
      A     L 0.1;
      JNB   _036;
      L     DB22.DBW 8200;
      T     DB21.DBW 6;
_036: NOP   0;
      A     L 0.1;
      JNB   _037;
      L     DB22.DBW 8202;
      T     DB21.DBW 8;
_037: NOP   0;
      A     L 0.1;
      JNB   _038;
      L     DB22.DBB 8844;
      T     DB21.DBB 476;
_038: NOP   0;
      A     L 0.0;
      A(;
      L     DB20.DBW 62;
      L     6;
      ==I;
      );
      =     L 0.1;
      A     L 0.1;
      JNB   _039;
      CALL  "BLKMOV" (
           SRCBLK                   := P#DB22.DBX 1600.0 DWORD 80,
           RET_VAL                  := MW 2044,
           DSTBLK                   := P#DB21.DBX 46.0 DWORD 80);
_039: NOP   0;
      A     L 0.1;
      JNB   _03a;
      L     DB22.DBW 8010;
      T     DB21.DBW 384;
_03a: NOP   0;
      A     L 0.1;
      JNB   _03b;
      L     DB22.DBD 6800;
      T     DB21.DBD 396;
_03b: NOP   0;
      A     L 0.1;
      JNB   _03c;
      L     DB22.DBD 6804;
      T     DB21.DBD 400;
_03c: NOP   0;
      A     L 0.1;
      JNB   _03d;
      L     DB22.DBW 8240;
      T     DB21.DBW 6;
_03d: NOP   0;
      A     L 0.1;
      JNB   _03e;
      L     DB22.DBW 8242;
      T     DB21.DBW 8;
_03e: NOP   0;
      A     L 0.1;
      JNB   _03f;
      L     DB22.DBB 8845;
      T     DB21.DBB 476;
_03f: NOP   0;
      A     L 0.0;
      A(;
      L     DB20.DBW 62;
      L     7;
      ==I;
      );
      =     L 0.1;
      A     L 0.1;
      JNB   _040;
      CALL  "BLKMOV" (
           SRCBLK                   := P#DB22.DBX 1920.0 DWORD 80,
           RET_VAL                  := MW 2044,
           DSTBLK                   := P#DB21.DBX 46.0 DWORD 80);
_040: NOP   0;
      A     L 0.1;
      JNB   _041;
      L     DB22.DBW 8012;
      T     DB21.DBW 384;
_041: NOP   0;
      A     L 0.1;
      JNB   _042;
      L     DB22.DBD 6880;
      T     DB21.DBD 396;
_042: NOP   0;
      A     L 0.1;
      JNB   _043;
      L     DB22.DBD 6884;
      T     DB21.DBD 400;
_043: NOP   0;
      A     L 0.1;
      JNB   _044;
      L     DB22.DBW 8280;
      T     DB21.DBW 6;
_044: NOP   0;
      A     L 0.1;
      JNB   _045;
      L     DB22.DBW 8282;
      T     DB21.DBW 8;
_045: NOP   0;
      A     L 0.1;
      JNB   _046;
      L     DB22.DBB 8846;
      T     DB21.DBB 476;
_046: NOP   0;
      A     L 0.0;
      A(;
      L     DB20.DBW 62;
      L     8;
      ==I;
      );
      =     L 0.1;
      A     L 0.1;
      JNB   _047;
      CALL  "BLKMOV" (
           SRCBLK                   := P#DB22.DBX 2240.0 DWORD 80,
           RET_VAL                  := MW 2044,
           DSTBLK                   := P#DB21.DBX 46.0 DWORD 80);
_047: NOP   0;
      A     L 0.1;
      JNB   _048;
      L     DB22.DBW 8014;
      T     DB21.DBW 384;
_048: NOP   0;
      A     L 0.1;
      JNB   _049;
      L     DB22.DBD 6960;
      T     DB21.DBD 396;
_049: NOP   0;
      A     L 0.1;
      JNB   _04a;
      L     DB22.DBD 6964;
      T     DB21.DBD 400;
_04a: NOP   0;
      A     L 0.1;
      JNB   _04b;
      L     DB22.DBW 8320;
      T     DB21.DBW 6;
_04b: NOP   0;
      A     L 0.1;
      JNB   _04c;
      L     DB22.DBW 8322;
      T     DB21.DBW 8;
_04c: NOP   0;
      A     L 0.1;
      JNB   _04d;
      L     DB22.DBB 8847;
      T     DB21.DBB 476;
_04d: NOP   0;
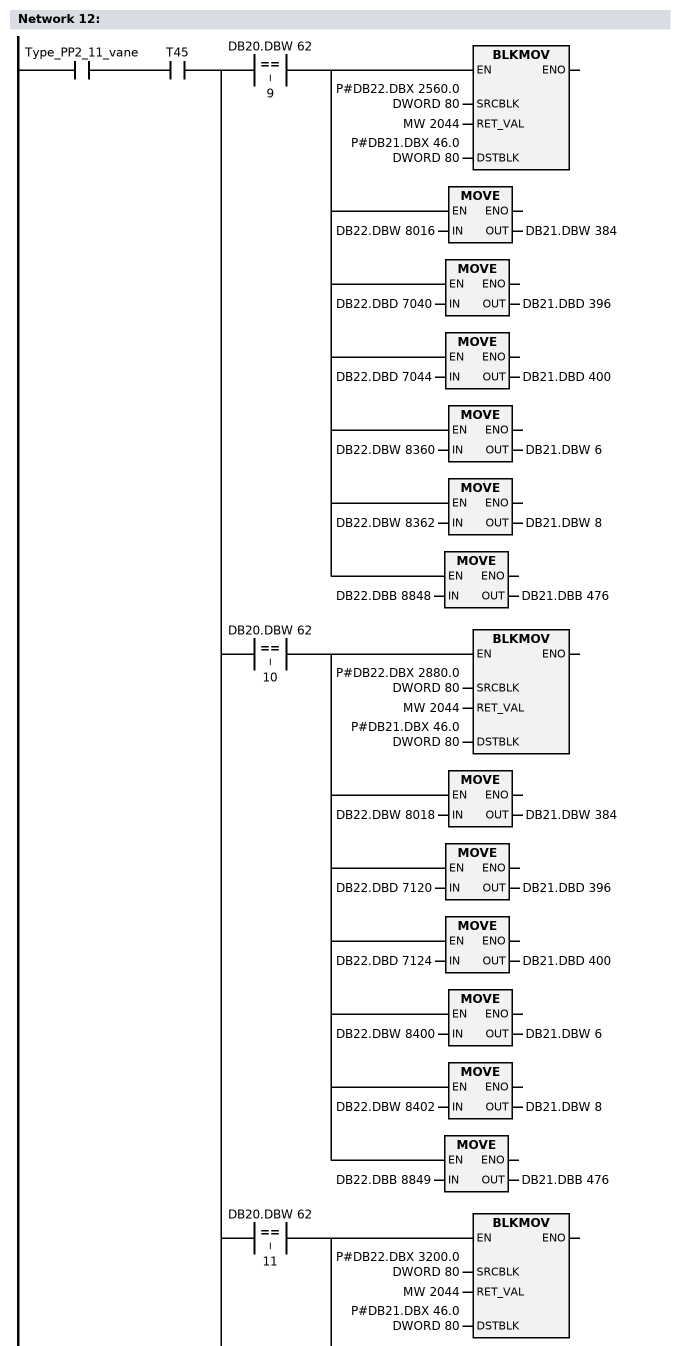
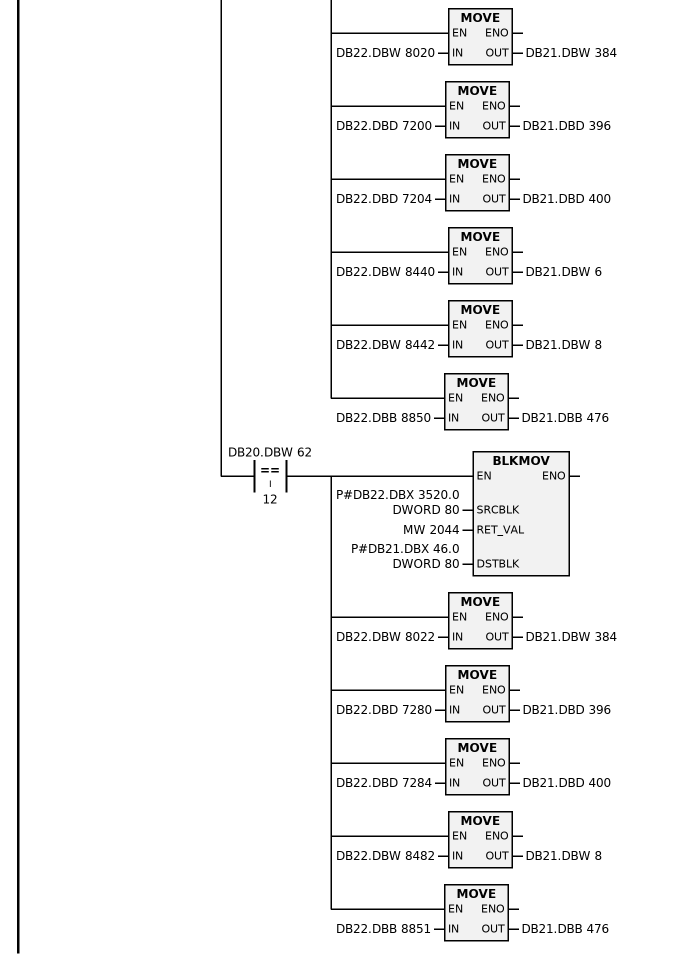
NETWORK
TITLE =
      A     "Type_PP2_11_vane";
      A     "T45";
      =     L 0.0;
      A     L 0.0;
      A(;
      L     DB20.DBW 62;
      L     9;
      ==I;
      );
      =     L 0.1;
      A     L 0.1;
      JNB   _04e;
      CALL  "BLKMOV" (
           SRCBLK                   := P#DB22.DBX 2560.0 DWORD 80,
           RET_VAL                  := MW 2044,
           DSTBLK                   := P#DB21.DBX 46.0 DWORD 80);
_04e: NOP   0;
      A     L 0.1;
      JNB   _04f;
      L     DB22.DBW 8016;
      T     DB21.DBW 384;
_04f: NOP   0;
      A     L 0.1;
      JNB   _050;
      L     DB22.DBD 7040;
      T     DB21.DBD 396;
_050: NOP   0;
      A     L 0.1;
      JNB   _051;
      L     DB22.DBD 7044;
      T     DB21.DBD 400;
_051: NOP   0;
      A     L 0.1;
      JNB   _052;
      L     DB22.DBW 8360;
      T     DB21.DBW 6;
_052: NOP   0;
      A     L 0.1;
      JNB   _053;
      L     DB22.DBW 8362;
      T     DB21.DBW 8;
_053: NOP   0;
      A     L 0.1;
      JNB   _054;
      L     DB22.DBB 8848;
      T     DB21.DBB 476;
_054: NOP   0;
      A     L 0.0;
      A(;
      L     DB20.DBW 62;
      L     10;
      ==I;
      );
      =     L 0.1;
      A     L 0.1;
      JNB   _055;
      CALL  "BLKMOV" (
           SRCBLK                   := P#DB22.DBX 2880.0 DWORD 80,
           RET_VAL                  := MW 2044,
           DSTBLK                   := P#DB21.DBX 46.0 DWORD 80);
_055: NOP   0;
      A     L 0.1;
      JNB   _056;
      L     DB22.DBW 8018;
      T     DB21.DBW 384;
_056: NOP   0;
      A     L 0.1;
      JNB   _057;
      L     DB22.DBD 7120;
      T     DB21.DBD 396;
_057: NOP   0;
      A     L 0.1;
      JNB   _058;
      L     DB22.DBD 7124;
      T     DB21.DBD 400;
_058: NOP   0;
      A     L 0.1;
      JNB   _059;
      L     DB22.DBW 8400;
      T     DB21.DBW 6;
_059: NOP   0;
      A     L 0.1;
      JNB   _05a;
      L     DB22.DBW 8402;
      T     DB21.DBW 8;
_05a: NOP   0;
      A     L 0.1;
      JNB   _05b;
      L     DB22.DBB 8849;
      T     DB21.DBB 476;
_05b: NOP   0;
      A     L 0.0;
      A(;
      L     DB20.DBW 62;
      L     11;
      ==I;
      );
      =     L 0.1;
      A     L 0.1;
      JNB   _05c;
      CALL  "BLKMOV" (
           SRCBLK                   := P#DB22.DBX 3200.0 DWORD 80,
           RET_VAL                  := MW 2044,
           DSTBLK                   := P#DB21.DBX 46.0 DWORD 80);
_05c: NOP   0;
      A     L 0.1;
      JNB   _05d;
      L     DB22.DBW 8020;
      T     DB21.DBW 384;
_05d: NOP   0;
      A     L 0.1;
      JNB   _05e;
      L     DB22.DBD 7200;
      T     DB21.DBD 396;
_05e: NOP   0;
      A     L 0.1;
      JNB   _05f;
      L     DB22.DBD 7204;
      T     DB21.DBD 400;
_05f: NOP   0;
      A     L 0.1;
      JNB   _060;
      L     DB22.DBW 8440;
      T     DB21.DBW 6;
_060: NOP   0;
      A     L 0.1;
      JNB   _061;
      L     DB22.DBW 8442;
      T     DB21.DBW 8;
_061: NOP   0;
      A     L 0.1;
      JNB   _062;
      L     DB22.DBB 8850;
      T     DB21.DBB 476;
_062: NOP   0;
      A     L 0.0;
      A(;
      L     DB20.DBW 62;
      L     12;
      ==I;
      );
      =     L 0.1;
      A     L 0.1;
      JNB   _063;
      CALL  "BLKMOV" (
           SRCBLK                   := P#DB22.DBX 3520.0 DWORD 80,
           RET_VAL                  := MW 2044,
           DSTBLK                   := P#DB21.DBX 46.0 DWORD 80);
_063: NOP   0;
      A     L 0.1;
      JNB   _064;
      L     DB22.DBW 8022;
      T     DB21.DBW 384;
_064: NOP   0;
      A     L 0.1;
      JNB   _065;
      L     DB22.DBD 7280;
      T     DB21.DBD 396;
_065: NOP   0;
      A     L 0.1;
      JNB   _066;
      L     DB22.DBD 7284;
      T     DB21.DBD 400;
_066: NOP   0;
      A     L 0.1;
      JNB   _067;
      L     DB22.DBW 8482;
      T     DB21.DBW 8;
_067: NOP   0;
      A     L 0.1;
      JNB   _068;
      L     DB22.DBB 8851;
      T     DB21.DBB 476;
_068: NOP   0;
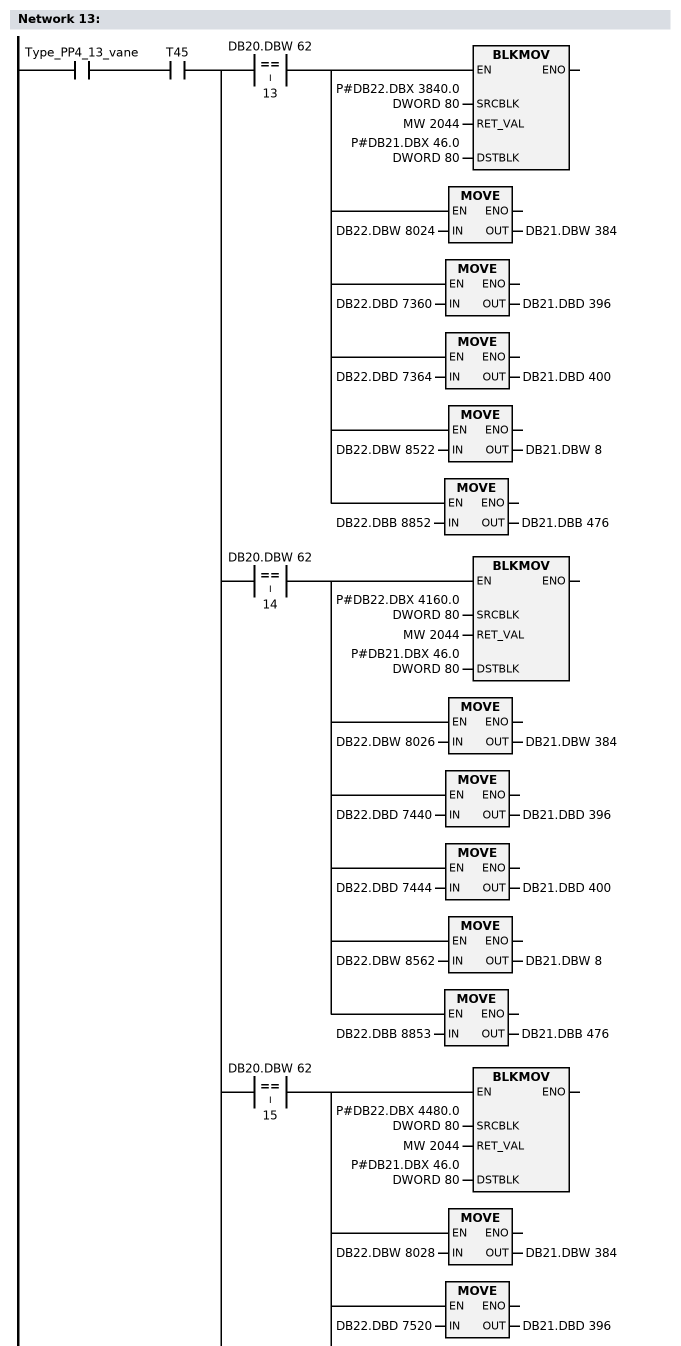
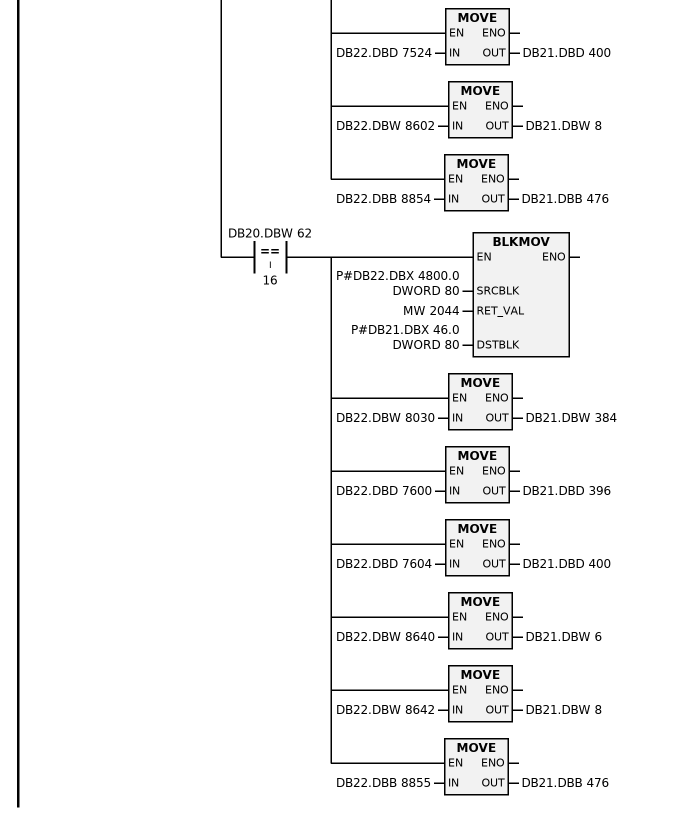
NETWORK
TITLE =
      A     "Type_PP4_13_vane";
      A     "T45";
      =     L 0.0;
      A     L 0.0;
      A(;
      L     DB20.DBW 62;
      L     13;
      ==I;
      );
      =     L 0.1;
      A     L 0.1;
      JNB   _069;
      CALL  "BLKMOV" (
           SRCBLK                   := P#DB22.DBX 3840.0 DWORD 80,
           RET_VAL                  := MW 2044,
           DSTBLK                   := P#DB21.DBX 46.0 DWORD 80);
_069: NOP   0;
      A     L 0.1;
      JNB   _06a;
      L     DB22.DBW 8024;
      T     DB21.DBW 384;
_06a: NOP   0;
      A     L 0.1;
      JNB   _06b;
      L     DB22.DBD 7360;
      T     DB21.DBD 396;
_06b: NOP   0;
      A     L 0.1;
      JNB   _06c;
      L     DB22.DBD 7364;
      T     DB21.DBD 400;
_06c: NOP   0;
      A     L 0.1;
      JNB   _06d;
      L     DB22.DBW 8522;
      T     DB21.DBW 8;
_06d: NOP   0;
      A     L 0.1;
      JNB   _06e;
      L     DB22.DBB 8852;
      T     DB21.DBB 476;
_06e: NOP   0;
      A     L 0.0;
      A(;
      L     DB20.DBW 62;
      L     14;
      ==I;
      );
      =     L 0.1;
      A     L 0.1;
      JNB   _06f;
      CALL  "BLKMOV" (
           SRCBLK                   := P#DB22.DBX 4160.0 DWORD 80,
           RET_VAL                  := MW 2044,
           DSTBLK                   := P#DB21.DBX 46.0 DWORD 80);
_06f: NOP   0;
      A     L 0.1;
      JNB   _070;
      L     DB22.DBW 8026;
      T     DB21.DBW 384;
_070: NOP   0;
      A     L 0.1;
      JNB   _071;
      L     DB22.DBD 7440;
      T     DB21.DBD 396;
_071: NOP   0;
      A     L 0.1;
      JNB   _072;
      L     DB22.DBD 7444;
      T     DB21.DBD 400;
_072: NOP   0;
      A     L 0.1;
      JNB   _073;
      L     DB22.DBW 8562;
      T     DB21.DBW 8;
_073: NOP   0;
      A     L 0.1;
      JNB   _074;
      L     DB22.DBB 8853;
      T     DB21.DBB 476;
_074: NOP   0;
      A     L 0.0;
      A(;
      L     DB20.DBW 62;
      L     15;
      ==I;
      );
      =     L 0.1;
      A     L 0.1;
      JNB   _075;
      CALL  "BLKMOV" (
           SRCBLK                   := P#DB22.DBX 4480.0 DWORD 80,
           RET_VAL                  := MW 2044,
           DSTBLK                   := P#DB21.DBX 46.0 DWORD 80);
_075: NOP   0;
      A     L 0.1;
      JNB   _076;
      L     DB22.DBW 8028;
      T     DB21.DBW 384;
_076: NOP   0;
      A     L 0.1;
      JNB   _077;
      L     DB22.DBD 7520;
      T     DB21.DBD 396;
_077: NOP   0;
      A     L 0.1;
      JNB   _078;
      L     DB22.DBD 7524;
      T     DB21.DBD 400;
_078: NOP   0;
      A     L 0.1;
      JNB   _079;
      L     DB22.DBW 8602;
      T     DB21.DBW 8;
_079: NOP   0;
      A     L 0.1;
      JNB   _07a;
      L     DB22.DBB 8854;
      T     DB21.DBB 476;
_07a: NOP   0;
      A     L 0.0;
      A(;
      L     DB20.DBW 62;
      L     16;
      ==I;
      );
      =     L 0.1;
      A     L 0.1;
      JNB   _07b;
      CALL  "BLKMOV" (
           SRCBLK                   := P#DB22.DBX 4800.0 DWORD 80,
           RET_VAL                  := MW 2044,
           DSTBLK                   := P#DB21.DBX 46.0 DWORD 80);
_07b: NOP   0;
      A     L 0.1;
      JNB   _07c;
      L     DB22.DBW 8030;
      T     DB21.DBW 384;
_07c: NOP   0;
      A     L 0.1;
      JNB   _07d;
      L     DB22.DBD 7600;
      T     DB21.DBD 396;
_07d: NOP   0;
      A     L 0.1;
      JNB   _07e;
      L     DB22.DBD 7604;
      T     DB21.DBD 400;
_07e: NOP   0;
      A     L 0.1;
      JNB   _07f;
      L     DB22.DBW 8640;
      T     DB21.DBW 6;
_07f: NOP   0;
      A     L 0.1;
      JNB   _080;
      L     DB22.DBW 8642;
      T     DB21.DBW 8;
_080: NOP   0;
      A     L 0.1;
      JNB   _081;
      L     DB22.DBB 8855;
      T     DB21.DBB 476;
_081: NOP   0;
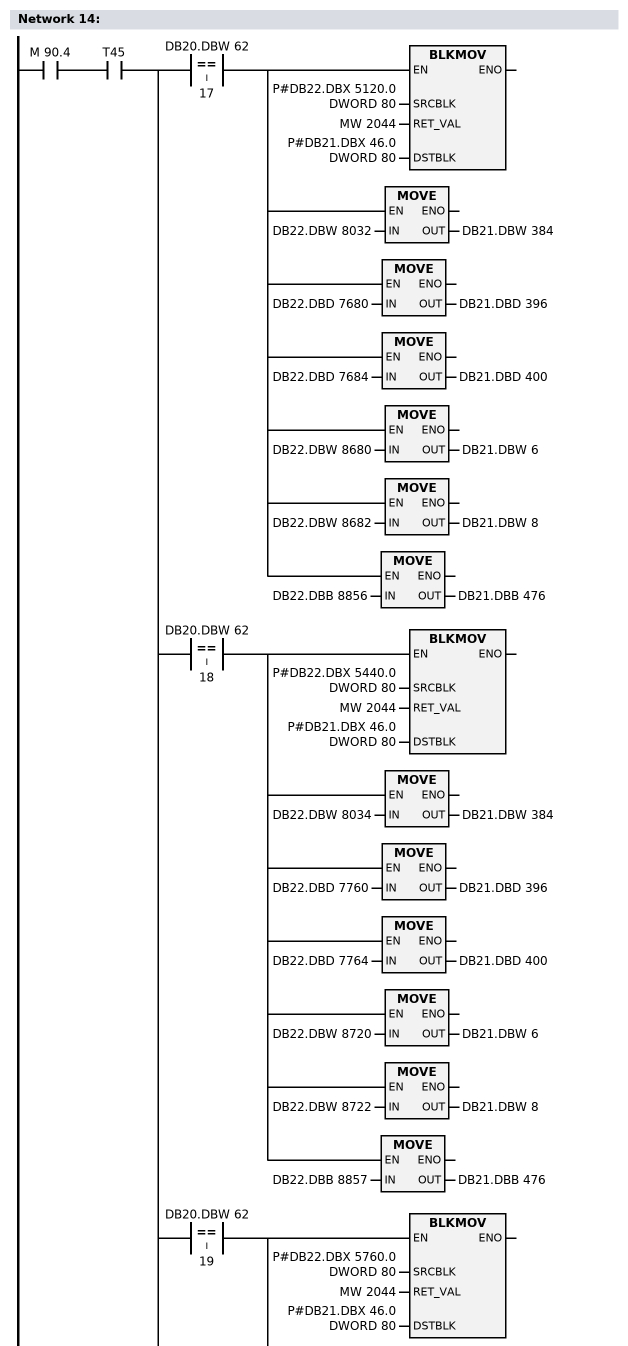
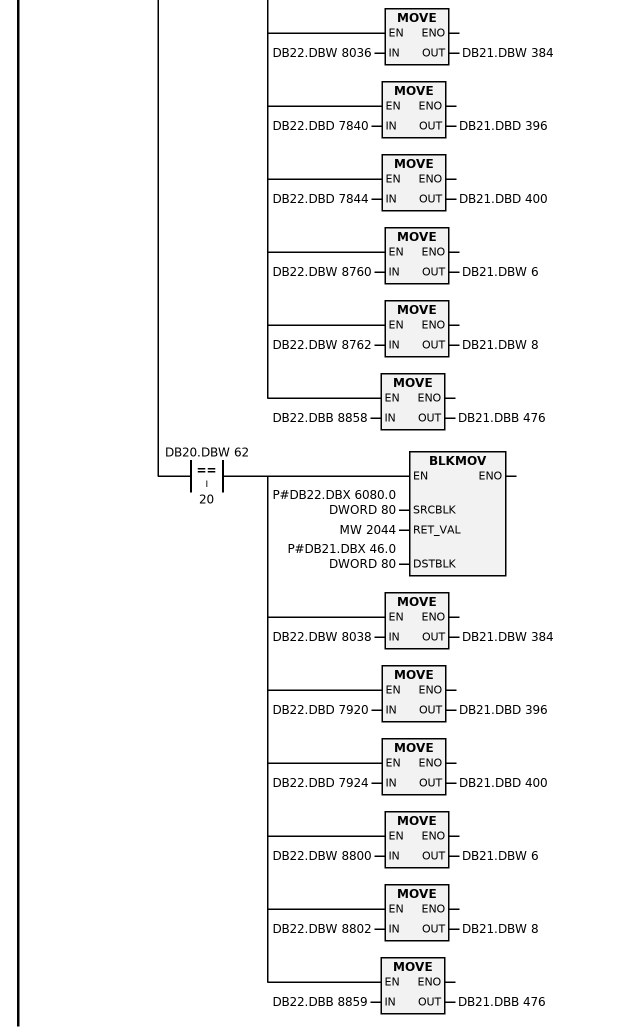
NETWORK
TITLE =
      A     M 90.4;
      A     "T45";
      =     L 0.0;
      A     L 0.0;
      A(;
      L     DB20.DBW 62;
      L     17;
      ==I;
      );
      =     L 0.1;
      A     L 0.1;
      JNB   _082;
      CALL  "BLKMOV" (
           SRCBLK                   := P#DB22.DBX 5120.0 DWORD 80,
           RET_VAL                  := MW 2044,
           DSTBLK                   := P#DB21.DBX 46.0 DWORD 80);
_082: NOP   0;
      A     L 0.1;
      JNB   _083;
      L     DB22.DBW 8032;
      T     DB21.DBW 384;
_083: NOP   0;
      A     L 0.1;
      JNB   _084;
      L     DB22.DBD 7680;
      T     DB21.DBD 396;
_084: NOP   0;
      A     L 0.1;
      JNB   _085;
      L     DB22.DBD 7684;
      T     DB21.DBD 400;
_085: NOP   0;
      A     L 0.1;
      JNB   _086;
      L     DB22.DBW 8680;
      T     DB21.DBW 6;
_086: NOP   0;
      A     L 0.1;
      JNB   _087;
      L     DB22.DBW 8682;
      T     DB21.DBW 8;
_087: NOP   0;
      A     L 0.1;
      JNB   _088;
      L     DB22.DBB 8856;
      T     DB21.DBB 476;
_088: NOP   0;
      A     L 0.0;
      A(;
      L     DB20.DBW 62;
      L     18;
      ==I;
      );
      =     L 0.1;
      A     L 0.1;
      JNB   _089;
      CALL  "BLKMOV" (
           SRCBLK                   := P#DB22.DBX 5440.0 DWORD 80,
           RET_VAL                  := MW 2044,
           DSTBLK                   := P#DB21.DBX 46.0 DWORD 80);
_089: NOP   0;
      A     L 0.1;
      JNB   _08a;
      L     DB22.DBW 8034;
      T     DB21.DBW 384;
_08a: NOP   0;
      A     L 0.1;
      JNB   _08b;
      L     DB22.DBD 7760;
      T     DB21.DBD 396;
_08b: NOP   0;
      A     L 0.1;
      JNB   _08c;
      L     DB22.DBD 7764;
      T     DB21.DBD 400;
_08c: NOP   0;
      A     L 0.1;
      JNB   _08d;
      L     DB22.DBW 8720;
      T     DB21.DBW 6;
_08d: NOP   0;
      A     L 0.1;
      JNB   _08e;
      L     DB22.DBW 8722;
      T     DB21.DBW 8;
_08e: NOP   0;
      A     L 0.1;
      JNB   _08f;
      L     DB22.DBB 8857;
      T     DB21.DBB 476;
_08f: NOP   0;
      A     L 0.0;
      A(;
      L     DB20.DBW 62;
      L     19;
      ==I;
      );
      =     L 0.1;
      A     L 0.1;
      JNB   _090;
      CALL  "BLKMOV" (
           SRCBLK                   := P#DB22.DBX 5760.0 DWORD 80,
           RET_VAL                  := MW 2044,
           DSTBLK                   := P#DB21.DBX 46.0 DWORD 80);
_090: NOP   0;
      A     L 0.1;
      JNB   _091;
      L     DB22.DBW 8036;
      T     DB21.DBW 384;
_091: NOP   0;
      A     L 0.1;
      JNB   _092;
      L     DB22.DBD 7840;
      T     DB21.DBD 396;
_092: NOP   0;
      A     L 0.1;
      JNB   _093;
      L     DB22.DBD 7844;
      T     DB21.DBD 400;
_093: NOP   0;
      A     L 0.1;
      JNB   _094;
      L     DB22.DBW 8760;
      T     DB21.DBW 6;
_094: NOP   0;
      A     L 0.1;
      JNB   _095;
      L     DB22.DBW 8762;
      T     DB21.DBW 8;
_095: NOP   0;
      A     L 0.1;
      JNB   _096;
      L     DB22.DBB 8858;
      T     DB21.DBB 476;
_096: NOP   0;
      A     L 0.0;
      A(;
      L     DB20.DBW 62;
      L     20;
      ==I;
      );
      =     L 0.1;
      A     L 0.1;
      JNB   _097;
      CALL  "BLKMOV" (
           SRCBLK                   := P#DB22.DBX 6080.0 DWORD 80,
           RET_VAL                  := MW 2044,
           DSTBLK                   := P#DB21.DBX 46.0 DWORD 80);
_097: NOP   0;
      A     L 0.1;
      JNB   _098;
      L     DB22.DBW 8038;
      T     DB21.DBW 384;
_098: NOP   0;
      A     L 0.1;
      JNB   _099;
      L     DB22.DBD 7920;
      T     DB21.DBD 396;
_099: NOP   0;
      A     L 0.1;
      JNB   _09a;
      L     DB22.DBD 7924;
      T     DB21.DBD 400;
_09a: NOP   0;
      A     L 0.1;
      JNB   _09b;
      L     DB22.DBW 8800;
      T     DB21.DBW 6;
_09b: NOP   0;
      A     L 0.1;
      JNB   _09c;
      L     DB22.DBW 8802;
      T     DB21.DBW 8;
_09c: NOP   0;
      A     L 0.1;
      JNB   _09d;
      L     DB22.DBB 8859;
      T     DB21.DBB 476;
_09d: NOP   0;
END_FUNCTION

FUNCTION "FC52 - SYSTEM VISION" : VOID	// FC 52
VERSION : 0.1
BEGIN
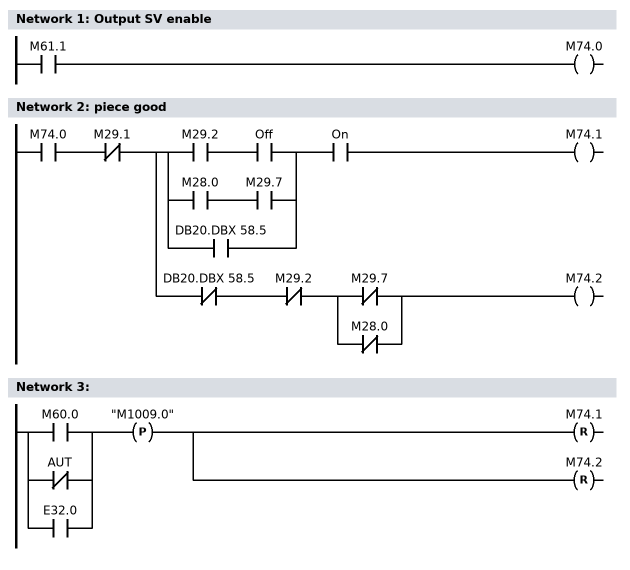
NETWORK
TITLE = Output SV enable
      A     "M61.1";
      =     "M74.0";
NETWORK
TITLE = piece good
      A     "M74.0";
      AN    "M29.1";
      =     L 0.0;
      A     L 0.0;
      A(;
      A     "M29.2";
      A     "Off";
      O;
      A     "M28.0";
      A     "M29.7";
      O     DB20.DBX 58.5;
      );
      A     "On";
      =     "M74.1";
      A     L 0.0;
      AN    DB20.DBX 58.5;
      AN    "M29.2";
      A(;
      ON    "M29.7";
      ON    "M28.0";
      );
      =     "M74.2";
NETWORK
TITLE =
      A(;
      O     "M60.0";
      ON    "AUT";
      O     "E32.0";
      );
      FP    "M1009.0";
      R     "M74.1";
      R     "M74.2";
END_FUNCTION

FUNCTION "FC53 - REWORK" : VOID	// FC 53
VERSION : 0.1
BEGIN
// (block stored without names or comments; labels and parameter names are numbered)
NETWORK
TITLE =
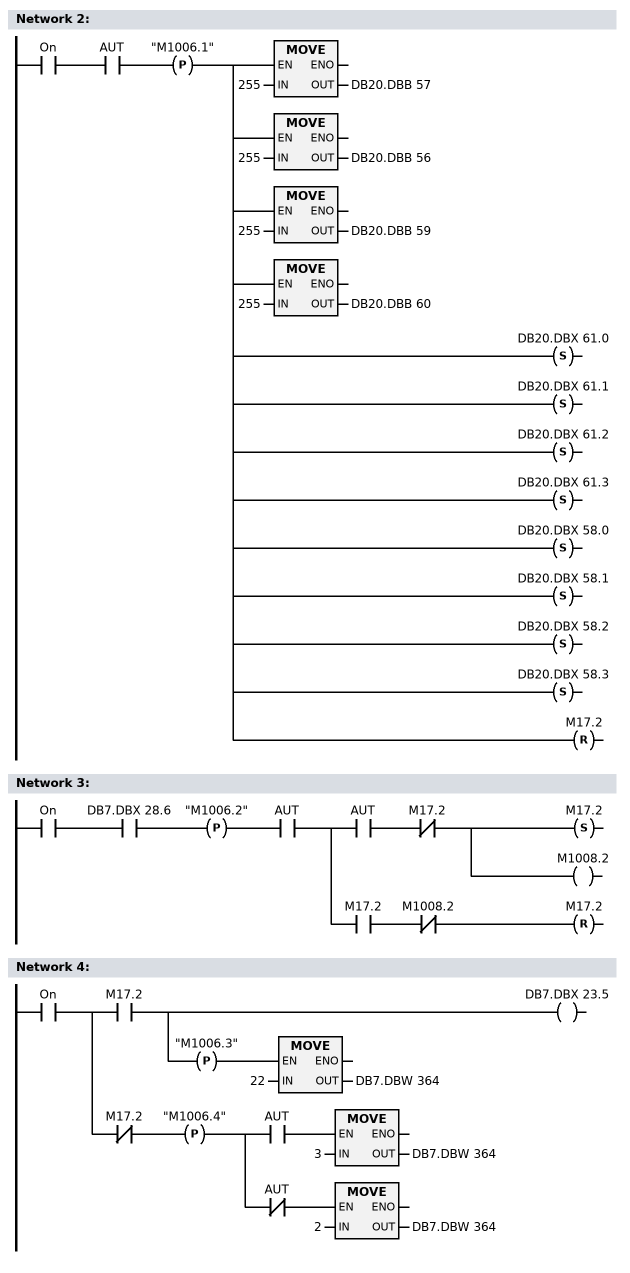
NETWORK
TITLE =
      A     "On";
      A     "AUT";
      FP    "M1006.1";
      =     L 0.0;
      A     L 0.0;
      JNB   M001;
      L     255;
      T     DB20.DBB 57;
M001: NOP   0;
      A     L 0.0;
      JNB   M002;
      L     255;
      T     DB20.DBB 56;
M002: NOP   0;
      A     L 0.0;
      JNB   M003;
      L     255;
      T     DB20.DBB 59;
M003: NOP   0;
      A     L 0.0;
      JNB   M004;
      L     255;
      T     DB20.DBB 60;
M004: NOP   0;
      A     L 0.0;
      BLD   102;
      S     DB20.DBX 61.0;
      A     L 0.0;
      BLD   102;
      S     DB20.DBX 61.1;
      A     L 0.0;
      BLD   102;
      S     DB20.DBX 61.2;
      A     L 0.0;
      BLD   102;
      S     DB20.DBX 61.3;
      A     L 0.0;
      BLD   102;
      S     DB20.DBX 58.0;
      A     L 0.0;
      BLD   102;
      S     DB20.DBX 58.1;
      A     L 0.0;
      BLD   102;
      S     DB20.DBX 58.2;
      A     L 0.0;
      BLD   102;
      S     DB20.DBX 58.3;
      A     L 0.0;
      BLD   102;
      R     "M17.2";
NETWORK
TITLE =
      A     "On";
      A     DB7.DBX 28.6;
      FP    "M1006.2";
      A     "AUT";
      =     L 0.0;
      A     L 0.0;
      A     "AUT";
      AN    "M17.2";
      S     "M17.2";
      =     "M1008.2";
      A     L 0.0;
      A     "M17.2";
      AN    "M1008.2";
      R     "M17.2";
NETWORK
TITLE =
      A     "On";
      =     L 0.0;
      A     L 0.0;
      A     "M17.2";
      =     L 0.1;
      A     L 0.1;
      BLD   102;
      =     DB7.DBX 23.5;
      A     L 0.1;
      FP    "M1006.3";
      JNB   M005;
      L     22;
      T     DB7.DBW 364;
M005: NOP   0;
      A     L 0.0;
      AN    "M17.2";
      FP    "M1006.4";
      =     L 0.1;
      A     L 0.1;
      A     "AUT";
      JNB   M006;
      L     3;
      T     DB7.DBW 364;
M006: NOP   0;
      A     L 0.1;
      AN    "AUT";
      JNB   M007;
      L     2;
      T     DB7.DBW 364;
M007: NOP   0;
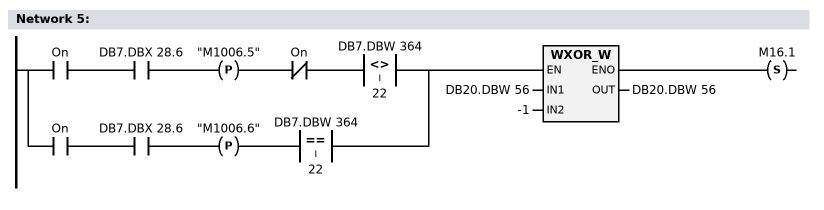
NETWORK
TITLE =
      A(;
      A     "On";
      A     DB7.DBX 28.6;
      FP    "M1006.5";
      AN    "On";
      A(;
      L     DB7.DBW 364;
      L     22;
      <>I;
      );
      O(;
      A     "On";
      A     DB7.DBX 28.6;
      FP    "M1006.6";
      A(;
      L     DB7.DBW 364;
      L     22;
      ==I;
      );
      );
      );
      JNB   M008;
      L     DB20.DBW 56;
      L     -1;
      XOW;
      T     DB20.DBW 56;
      SET;
      SAVE;
      CLR;
M008: A     BR;
      S     "M16.1";
